CASE DP_Step3 OF 
100://负极叠片，正极在取片位
	bStandbyStep1_1:=FALSE;
	bStandbyStep1_2:=FALSE;
	DP_Step3:=110; 
110:   //叠负极片同时 判断证据能否取片  提高效率
	IF arrAxisCtrl[AxiseNo.VirAxisName.VirMain].Status.fActPos>=10  AND  arrAxisCtrl[AxiseNo.VirAxisName.VirMain].Status.fActPos<=220     THEN
	//正送片搬运极取片处理
		IF   arrAxisCtrl[AxiseNo.AxisName.AnCarryingUpDown].Cmd.arrbRealPoint[4] AND 
			  NOT Mach_Control.An_b.An_CarryingFalg    AND  ( Mach_Control.An_b.An_MainBeltOK OR  Mach_Control.U.EmptyRunMode )  AND 
			  NOT  Mach_Control.An_b.An_MainBelting   AND NOT  bStandbyStep1_1 AND (NOT An_JumpRules[3]  AND NOT  An_JumpRules[6] AND NOT An_JumpRules[8] AND NOT An_JumpRules[10])(*AND NOT Mach_Control.An_b.JumpPiceReady *) THEN
			   An_Step0:=10;//正极取流水线子程序
			   bStandbyStep1_1:=TRUE;
		END_IF
		
		IF arrAxisCtrl[AxiseNo.AxisName.AnDTCarryingUpDown].Cmd.arrbRealPoint[4] AND 
		 Mach_Control.An_b.An_deviationDPOK AND NOT Mach_Control.An_b.An_DPCarryingFalg AND  
			Mach_Control.An_b.An_deviationFalg  AND  NOT  bStandbyStep1_2  AND NOT DP_CheseCam  THEN
			An_Step3:=10;//正极取纠偏平台子程序
			bStandbyStep1_2:=TRUE;
		END_IF
	
	ELSIF  arrAxisCtrl[AxiseNo.VirAxisName.VirMain].Status.fActPos>220  THEN
		DP_Step3:=120;
	END_IF		   
	
	
120:
	arrCyCtrl[arrCyNo.ElectValveName.CadeviationVacuum].Cmd.bON:=TRUE;//负极纠偏平台真空开			
	arrCyCtrl[arrCyNo.ElectValveName.CadeviationVacuum].Cmd.bOFF:=FALSE;//负极纠偏平台真空开					
	IF 	arrAxisCtrl[AxiseNo.VirAxisName.VirMain].Status.fActPos>=234 THEN//198
		
		Mach_Control.Ca_b.Ca_Rectifydev_CS:=0;
		CCD.Over.Start.stPoleNo:=Par.stDT_date.Ca_MQ_Slice[8].stPoleNo;
		arrCyCtrl[arrCyNo.ElectValveName.CaDTCarryingVacuum].Cmd.bON:=TRUE;//负极叠片搬运真空破
		arrCyCtrl[arrCyNo.ElectValveName.CaDTCarryingVacuum].Cmd.bOFF:=FALSE;//负极叠片搬运真空破
		arrCyCtrl[arrCyNo.ElectValveName.CaCarryingVacuum2].Cmd.bON:=TRUE;//负极送片搬运真空破
		arrCyCtrl[arrCyNo.ElectValveName.CaCarryingVacuum2].Cmd.bOFF:=FALSE;//负极送片搬运真空破
		arrCyCtrl[arrCyNo.ElectValveName.CadeviationVacuum].Cmd.bON:=TRUE;//负极纠偏平台真空开
		arrCyCtrl[arrCyNo.ElectValveName.CadeviationVacuum].Cmd.bOFF:=FALSE;//负极纠偏平台真空开			
		
		Mach_Control.Ca_b.Ca_DPCarryingFalg :=FALSE;//复位负极叠片搬运吸盘上有料标记
		//IF Mach_Control.Ca_b.Ca_CarryingFalg THEN
			Mach_Control.Ca_b.Ca_deviationFalg:=TRUE;//置位纠偏平台上有料标记
			Mach_Control.Ca_b.Ca_CarryingFalg:=FALSE;//复位负极送片搬运吸盘上有料标记
		//END_IF
		Par.stDT_date.Ca_MQ_Slice[8]:=Par.stDT_date.Ca_MQ_Slice[7];
		
	END_IF	
	IF 	arrAxisCtrl[AxiseNo.VirAxisName.VirMain].Status.fActPos>=342 THEN//198
     	CCD.Over.Start.iPliesNo:=UINT_TO_INT(Mach_Control.Ca_b.Ca_Quantited + Mach_Control.An_b.An_Quantited+1);	
		IF NOT Ca_Number THEN
			CCD.Over.Start.iPhotoDo:=1;
		ELSE
			CCD.Over.Start.iPhotoDo:=2;
		END_IF
		Mach_Control.DT_b.CDD_OverStart:=TRUE;
		DP_Step3:=121;
	 END_IF		
		
121:
	IF 	arrAxisCtrl[AxiseNo.VirAxisName.VirMain].Status.fActPos>=360 THEN//198
		arrCyCtrl[arrCyNo.ElectValveName.CaCarryingVacuum2].Cmd.bON:=FALSE;//负极送片搬运真空开
		arrCyCtrl[arrCyNo.ElectValveName.CaCarryingVacuum2].Cmd.bOFF:=TRUE;//负极送片搬运真空开
		arrCyCtrl[arrCyNo.ElectValveName.CaDTCarryingVacuum].Cmd.bON:=FALSE;//负极叠片搬运真空破
		arrCyCtrl[arrCyNo.ElectValveName.CaDTCarryingVacuum].Cmd.bOFF:=TRUE;//负极叠片搬运真空破
		DP_Step3:=6666;
	END_IF	
	
	
200://负极叠片，正极在取片位

	IF iAnCamInSel2=1 THEN
		arrCyCtrl[arrCyNo.ElectValveName.AnDTCarryingVacuum].Cmd.bON:=TRUE;//正极送片搬运真空关
		arrCyCtrl[arrCyNo.ElectValveName.AnDTCarryingVacuum].Cmd.bOFF:=FALSE;//正极送片搬运真空关
	END_IF
	
	//fbAnDTCarryingVacuum.Vacuumsel:=SEL(iAnCamInSel2=1,0,1)     ;//	正极叠片搬运真空开	
	IF arrAxisCtrl[AxiseNo.VirAxisName.VirMain].Status.fActPos>=210 THEN//复检提前
		IF Mach_Control.DT_b.DT_CCD_TwoModel THEN												
			CCD.AnRec.Finish.RectifyResult:=0;
			CCD.AnRec.Finish.RectifyX1:=0;
			CCD.AnRec.Finish.RectifyX2:=0;
			CCD.AnRec.Finish.RectifyY:=0;												
			Mach_Control.An_b.An_CCDStart :=TRUE;//启动CCD拍照
			CCD.AnRec.Start.iPhotoDo:=2;//第二次拍照	
		END_IF
		DP_Step3:=205;
	END_IF
205:			
	IF NOT DP_CheseCam  AND NOT  An_JumpRules[3]  AND NOT  An_JumpRules[6] AND NOT An_JumpRules[8] AND NOT An_JumpRules[10] THEN
	
		IF arrAxisCtrl[AxiseNo.VirAxisName.VirMain].Status.fActPos>=225  AND arrAxisCtrl[AxiseNo.VirAxisName.VirMain].Status.fActPos<=230 THEN	
			//fbAnCamInCarryingUpDown.bCamInExecute:=FALSE;//正极升解除耦合															
			//fbAnCamInCarryingWhirling.bCamInExecute:=FALSE;//正极旋转解除耦合			
			//Mach_Control.An_b.An_MainBelting:=FALSE;//正极搬运升降取极片中																					
			IF  NOT  Mach_Control.Ca_b.Ca_deviationFPOK  THEN    //负极放片纠偏太未在初始位置报警  
					Mach_Control.Ca_b.Error_tips[1]:=TRUE ;
			END_IF											
			IF  NOT  Mach_Control.An_b.An_deviationDPOK  THEN    //正极取片纠偏未完成报警
					Mach_Control.An_b.Error_tips[1]:=TRUE;
			END_IF			
			IF Mach_Control.An_b.An_deviationDPOK OR Mach_Control.U.EmptyRunMode OR	TRUE  THEN // 
				arrCyCtrl[arrCyNo.ElectValveName.AnDTCarryingVacuum].Cmd.bON:=TRUE;//正极叠片搬运真空开	
				arrCyCtrl[arrCyNo.ElectValveName.AnDTCarryingVacuum].Cmd.bOFF:=FALSE;//正极叠片搬运真空开		
				An_deviationDPOKFalg:=TRUE;	
			ELSE		
				arrCyCtrl[arrCyNo.ElectValveName.AnDTCarryingVacuum].Cmd.bON:=FALSE;//正极叠片搬运真空开					
				arrCyCtrl[arrCyNo.ElectValveName.AnDTCarryingVacuum].Cmd.bOFF:=TRUE;//正极叠片搬运真空开												
				fbAnCamInDTCarryingUpDown.bCamInExecute:=FALSE;	//正极叠片搬运升降凸轮解耦				
				IF NOT arrAxisCtrl[AxiseNo.AxisName.AnDTCarryingUpDown].Cmd.arrbRealPoint[4]    THEN
						arrAxisCtrl[AxiseNo.AxisName.AnDTCarryingUpDown].Cmd.iGoSetPos:=4;   //到等待位
				END_IF			
			END_IF	
			//IF NOT Mach_Control.An_b.JumpPiceReady THEN
				An_Step0:=10;//调用正极取片程序	
			//END_IF
			DP_Step3:=210;														
		END_IF									
	ELSE
			DP_Step3:=210;	
	END_IF


210:
	//打开或关闭真空，标记对应位置有料
	IF 	arrAxisCtrl[AxiseNo.VirAxisName.VirMain].Status.fActPos>=234 THEN//198
	
		Mach_Control.Ca_b.Ca_Rectifydev_CS:=0;
		arrCyCtrl[arrCyNo.ElectValveName.CaCarryingVacuum2].Cmd.bON:=TRUE;//负极送片搬运真空关
		arrCyCtrl[arrCyNo.ElectValveName.CaCarryingVacuum2].Cmd.bOFF:=FALSE;//负极送片搬运真空关
		arrCyCtrl[arrCyNo.ElectValveName.CaDTCarryingVacuum].Cmd.bON:=TRUE;//负极叠片搬运直空关
		arrCyCtrl[arrCyNo.ElectValveName.CaDTCarryingVacuum].Cmd.bOFF:=FALSE;//负极叠片搬运直空关
		arrCyCtrl[arrCyNo.ElectValveName.CadeviationVacuum].Cmd.bON:=TRUE;//负极纠偏平台真空开	
		arrCyCtrl[arrCyNo.ElectValveName.CadeviationVacuum].Cmd.bOFF:=FALSE;//负极纠偏平台真空开		
		
		Mach_Control.Ca_b.Ca_DPCarryingFalg :=FALSE;//复位负极叠片搬运吸盘上有料标记
		//IF Mach_Control.Ca_b.Ca_CarryingFalg THEN
			Mach_Control.Ca_b.Ca_deviationFalg:=TRUE;//置位纠偏平台上有料标记
			Mach_Control.Ca_b.Ca_CarryingFalg:=FALSE;//复位负极送片搬运吸盘上有料标记
		//END_IF
		Par.stDT_date.Ca_MQ_Slice[8]:=Par.stDT_date.Ca_MQ_Slice[7];
		IF An_deviationDPOKFalg AND  iAnCamInSel2=1   THEN
			Par.stDT_date.An_MQ_Slice[2]:=Par.stDT_date.An_MQ_Slice[1];
			//IF Mach_Control.An_b.An_deviationFalg THEN
				Mach_Control.An_b.An_DPCarryingFalg :=TRUE;//复位正极叠片搬运吸盘上有料标记										
				Mach_Control.An_b.An_deviationFalg:=FALSE;//置位纠偏平台上有料标记	
			//END_IF										
			arrCyCtrl[arrCyNo.ElectValveName.AndeviationVacuum].Cmd.bOFF:=TRUE;//正极纠偏平台真空关
			arrCyCtrl[arrCyNo.ElectValveName.AndeviationVacuum].Cmd.bON:=FALSE;//正极纠偏平台真空关
			arrCyCtrl[arrCyNo.ElectValveName.AndeviationVacuumBark].Cmd.bON:=TRUE;//正极纠偏平台破真空开	
			arrCyCtrl[arrCyNo.ElectValveName.AndeviationVacuumBark].Cmd.bOFF:=FALSE;//正极纠偏平台破真空开	
	(*	
		ELSIF NOT   DP_CheseCam THEN								
			An_Step3:=10;//正极叠片搬运取纠偏台极片	
	*)																					
		END_IF
	
	END_IF

	IF 	arrAxisCtrl[AxiseNo.VirAxisName.VirMain].Status.fActPos>=342 THEN//198
		CCD.Over.Start.iPliesNo:=UINT_TO_INT(Mach_Control.Ca_b.Ca_Quantited + Mach_Control.An_b.An_Quantited+1);
		CCD.Over.Start.stPoleNo:=Par.stDT_date.Ca_MQ_Slice[8].stPoleNo;
		IF NOT Ca_Number THEN
			CCD.Over.Start.iPhotoDo:=1;
		ELSE
			CCD.Over.Start.iPhotoDo:=2;
		END_IF
		Mach_Control.DT_b.CDD_OverStart:=TRUE;	
		IF NOT Ca_Number THEN
			DP_Step3:=211;					
		END_IF	
    END_IF	
211:
	IF 	arrAxisCtrl[AxiseNo.VirAxisName.VirMain].Status.fActPos>=360 THEN//198	
		arrCyCtrl[arrCyNo.ElectValveName.CaCarryingVacuum2].Cmd.bON:=FALSE;//负极送片搬运真空开
		arrCyCtrl[arrCyNo.ElectValveName.CaCarryingVacuum2].Cmd.bOFF:=TRUE;//负极送片搬运真空开
		arrCyCtrl[arrCyNo.ElectValveName.CaDTCarryingVacuum].Cmd.bON:=FALSE;//负极叠片搬运直空开
		arrCyCtrl[arrCyNo.ElectValveName.CaDTCarryingVacuum].Cmd.bOFF:=TRUE;//负极叠片搬运直空开
		DP_Step3:=6666;					
	END_IF
			



		
300://正极叠片，负极在取片位			
	bStandbyStep1_3:=FALSE;
	bStandbyStep1_4:=FALSE;
	DP_Step3:=310; 		
310:	
	IF arrAxisCtrl[AxiseNo.VirAxisName.VirMain].Status.fActPos>=10  AND  arrAxisCtrl[AxiseNo.VirAxisName.VirMain].Status.fActPos<=220     THEN
		//正送片搬运极取片处理
		IF   arrAxisCtrl[AxiseNo.AxisName.CaCarryingUpDown2].Cmd.arrbRealPoint[4] AND 
			NOT Mach_Control.Ca_b.Ca_CarryingFalg    AND  ( Mach_Control.Ca_b.Ca_CacheBeltDLOK OR  Mach_Control.U.EmptyRunMode )  AND 
			NOT  Mach_Control.Ca_b.Ca_CacheBelting   AND NOT  bStandbyStep1_3 THEN
			Ca_Step0:=10;   //负极取流水线子程序
			bStandbyStep1_3:=TRUE;
		END_IF
	
		IF arrAxisCtrl[AxiseNo.AxisName.CaDTCarryingUpDown].Cmd.arrbRealPoint[4] AND 
			Mach_Control.Ca_b.Ca_deviationDPOK AND NOT Mach_Control.Ca_b.Ca_DPCarryingFalg AND  
			Mach_Control.Ca_b.Ca_deviationFalg AND  NOT  bStandbyStep1_4   THEN
			Ca_Step3:=10;     //负极取纠偏平台子程序
			bStandbyStep1_4:=TRUE;
		END_IF					
	ELSIF  arrAxisCtrl[AxiseNo.VirAxisName.VirMain].Status.fActPos>220  THEN
			DP_Step3:=320; 
	END_IF	
	
320://正极叠片，负极在取片位
	arrCyCtrl[arrCyNo.ElectValveName.AndeviationVacuum].Cmd.bON:=TRUE;//正极纠偏平台真空开			
	arrCyCtrl[arrCyNo.ElectValveName.AndeviationVacuum].Cmd.bOFF:=FALSE;//正极纠偏平台真空开					
	IF 	arrAxisCtrl[AxiseNo.VirAxisName.VirMain].Status.fActPos>=234 THEN//198
	
		Mach_Control.An_b.An_Rectifydev_CS:=0;	
		arrCyCtrl[arrCyNo.ElectValveName.AnCarryingVacuum].Cmd.bON:=FALSE;//正极送片搬运真空关
		arrCyCtrl[arrCyNo.ElectValveName.AnCarryingVacuum].Cmd.bOFF:=TRUE;//正极送片搬运真空关
		arrCyCtrl[arrCyNo.ElectValveName.AnCarryingVacuumBark].Cmd.bON:=TRUE;//正极送片搬运破真空开
		arrCyCtrl[arrCyNo.ElectValveName.AnCarryingVacuumBark].Cmd.bOFF:=FALSE;//正极送片搬运破真空开
		
		arrCyCtrl[arrCyNo.ElectValveName.AnDTCarryingVacuum].Cmd.bON:=FALSE;//正极送片搬运真空关
		arrCyCtrl[arrCyNo.ElectValveName.AnDTCarryingVacuum].Cmd.bOFF:=TRUE;//正极送片搬运真空关
		arrCyCtrl[arrCyNo.ElectValveName.AnDTCarryingVacuumBark].Cmd.bON:=TRUE;//正极送片搬运破真空开
		arrCyCtrl[arrCyNo.ElectValveName.AnDTCarryingVacuumBark].Cmd.bOFF:=FALSE;//正极送片搬运破真空开
		
		arrCyCtrl[arrCyNo.ElectValveName.AndeviationVacuum].Cmd.bON:=TRUE;//正极纠偏平台真空开		
		arrCyCtrl[arrCyNo.ElectValveName.AndeviationVacuum].Cmd.bOFF:=FALSE;//正极纠偏平台真空开		
		
		
		Mach_Control.An_b.An_DPCarryingFalg :=FALSE;//复位正极叠片搬运吸盘上有料标记
		//IF Mach_Control.An_b.An_CarryingFalg THEN
			Mach_Control.An_b.An_deviationFalg:=TRUE;//置位纠偏平台上有料标记
			Mach_Control.An_b.An_CarryingFalg:=FALSE;//复位正极送片搬运吸盘上有料标记
		//END_IF
		Par.stDT_date.An_MQ_Slice[1]:=Par.stDT_date.An_MQ_Slice[0];
		
	END_IF
	
	IF 	arrAxisCtrl[AxiseNo.VirAxisName.VirMain].Status.fActPos>=342 THEN//198
		CCD.Over.Start.iPliesNo:=UINT_TO_INT(Mach_Control.Ca_b.Ca_Quantited + Mach_Control.An_b.An_Quantited+1);
		CCD.Over.Start.stPoleNo:=Par.stDT_date.An_MQ_Slice[2].stPoleNo;
		IF NOT An_Number THEN
			CCD.Over.Start.iPhotoDo:=1;
		ELSE
			CCD.Over.Start.iPhotoDo:=2;
		END_IF
		Mach_Control.DT_b.CDD_OverStart:=TRUE;				
		DP_Step3:=6666;	
	END_IF
400:	//复检提前------//正极叠片，负极在叠片位

	//fbCaDTCarryingVacuum.Vacuumsel:= SEL(iCaCamInSel2=1 ,0,1)   ;//	负极叠片搬运真空开
	IF iCaCamInSel2=1 THEN
		arrCyCtrl[arrCyNo.ElectValveName.CaDTCarryingVacuum].Cmd.bON:=FALSE;//负极叠台搬运真空开	
		arrCyCtrl[arrCyNo.ElectValveName.CaDTCarryingVacuum].Cmd.bOFF:=TRUE;//负极叠台搬运真空开		
	END_IF

	IF 	arrAxisCtrl[AxiseNo.VirAxisName.VirMain].Status.fActPos>=210 THEN//198
		IF Mach_Control.DT_b.DT_CCD_TwoModel THEN
				CCD.CaRec.Finish.RectifyX1:=0;
				CCD.CaRec.Finish.RectifyX2:=0;
				CCD.CaRec.Finish.RectifyY:=0;		
				CCD.CaRec.Finish.RectifyResult:=0;//拍照结果清零									
				Mach_Control.Ca_b.Ca_CCDStart :=TRUE;//启动CCD拍照
				CCD.CaRec.Start.iPhotoDo:=2;//启动CCD第二次拍照									
		END_IF
		DP_Step3:=405;
	END_IF
405:		
	IF arrAxisCtrl[AxiseNo.VirAxisName.VirMain].Status.fActPos>=225  AND arrAxisCtrl[AxiseNo.VirAxisName.VirMain].Status.fActPos<=230 THEN																								
		IF  NOT  Mach_Control.An_b.An_deviationFPOK  THEN    //正极放片纠偏太未在初始位置报警  
			  Mach_Control.An_b.Error_tips[2]:=TRUE ;
		END_IF
		
		IF  NOT  Mach_Control.Ca_b.Ca_deviationDPOK  THEN    //负极取片纠偏未完成报警
			  Mach_Control.Ca_b.Error_tips[2]:=TRUE ;
		END_IF		

		//正极叠片时平移到位后判断正极纠偏台是否允许放片
		IF Mach_Control.An_b.An_deviationFPOK OR Mach_Control.U.EmptyRunMode  THEN 
				An_deviationFPOKFalg:=TRUE;//正极纠偏平台允许放片标记
		ELSE									
			fbAnCamInCarryingUpDown.bCamInExecute:=FALSE;	//正极送片搬运升降凸轮解耦				
			IF NOT arrAxisCtrl[AxiseNo.AxisName.AnCarryingUpDown].Cmd.arrbRealPoint[4]    THEN
				arrAxisCtrl[AxiseNo.AxisName.AnCarryingUpDown].Cmd.iGoSetPos:=4;
			END_IF;				
		END_IF					
		IF Mach_Control.Ca_b.Ca_deviationDPOK OR Mach_Control.U.EmptyRunMode OR TRUE  THEN //  
			Ca_deviationDPOKFalg:=TRUE;	
			arrCyCtrl[arrCyNo.ElectValveName.CaDTCarryingVacuum].Cmd.bON:=FALSE;//负极叠片搬运真空开	
			arrCyCtrl[arrCyNo.ElectValveName.CaDTCarryingVacuum].Cmd.bOFF:=TRUE;//负极叠片搬运真空开		
		ELSE	
			//arrCyCtrl[arrCyNo.ElectValveName.CaDTCarryingVacuum].Cmd.bON:=FALSE;//负极叠片搬运真空开									
			fbCaCamInDTCarryingUpDown.bCamInExecute:=FALSE;	//负极叠片搬运升降凸轮解耦				
			IF NOT arrAxisCtrl[AxiseNo.AxisName.CaDTCarryingUpDown].Cmd.arrbRealPoint[4]    THEN
				arrAxisCtrl[AxiseNo.AxisName.CaDTCarryingUpDown].Cmd.iGoSetPos:=4;   //到等待位
			ELSE
				arrAxisCtrl[AxiseNo.AxisName.CaDTCarryingUpDown].Cmd.iGoSetPos:=0;   //到等待位
			END_IF;				
		END_IF									
		Ca_Step0:=10;//调用负极取片程序       取片允许条件在子程序里
		DP_Step3:=410;		
	END_IF
(*	
	//判断是否允许负极送片搬运取料
	IF arrAxisCtrl[AxiseNo.VirAxisName.VirMain].Status.fActPos>=CamOutArgel  AND arrAxisCtrl[AxiseNo.VirAxisName.VirMain].Status.fActPos<=(CamOutArgel+5) THEN
		IF (Mach_Control.Ca_b.Ca_CacheBeltDLOK AND NOT fbCaCamInCarryingUpDown2OutCamFlge) OR Mach_Control.U.EmptyRunMode  THEN
			Mach_Control.Ca_b.Ca_CacheBelting:=TRUE;//f负极搬运升降取极片中	
			arrCyCtrl[arrCyNo.ElectValveName.CaCarryingVacuum2].Cmd.bON:=FALSE;//负极送片搬运真空开
			arrCyCtrl[arrCyNo.ElectValveName.CaCarryingVacuum2].Cmd.bOFF:=TRUE;//负极送片搬运真空开
		ELSE
			//arrCyCtrl[arrCyNo.ElectValveName.CaCarryingVacuum2].Cmd.bON:=FALSE;//负极送片搬运真空开
			fbCaCamInCarryingUpDown2.bCamInExecute:=FALSE;//负极升解除耦合
			Mach_Control.Ca_b.Ca_CacheBelting:=FALSE;
		END_IF								
	END_IF
	//解除负极搬运升降凸轮耦合标记
	fbCaCamInCarryingUpDown2OutCam_F_TRIG(CLK:=fbCaCamInCarryingUpDown2.bCamInExecute , Q=> );
	IF fbCaCamInCarryingUpDown2OutCam_F_TRIG.Q THEN
		fbCaCamInCarryingUpDown2OutCamFlge:=TRUE;//负极升降2凸轮解耦标记
	END_IF	
*)			
410:							
	//打开或关闭真空，标记对应位置有料
	IF 	arrAxisCtrl[AxiseNo.VirAxisName.VirMain].Status.fActPos>=234 THEN//198

		Mach_Control.An_b.An_Rectifydev_CS:=0;
		CCD.Over.Start.stPoleNo:=Par.stDT_date.An_MQ_Slice[2].stPoleNo;
	(*	
		arrCyCtrl[arrCyNo.ElectValveName.AnCarryingVacuum].Cmd.bOFF:=TRUE;//正极送片搬运真空关
		arrCyCtrl[arrCyNo.ElectValveName.AnCarryingVacuumBark].Cmd.bON:=TRUE;//正极送片搬运破真空开
		arrCyCtrl[arrCyNo.ElectValveName.AnDTCarryingVacuum].Cmd.bOFF:=TRUE;//正极叠片搬运真空关
		arrCyCtrl[arrCyNo.ElectValveName.AnDTCarryingVacuumBark].Cmd.bON:=TRUE;//正极叠片搬运破真空开
	*)	
		arrCyCtrl[arrCyNo.ElectValveName.AnCarryingVacuum].Cmd.bON:=FALSE;//正极送片搬运真空关
		arrCyCtrl[arrCyNo.ElectValveName.AnCarryingVacuum].Cmd.bOFF:=TRUE;//正极送片搬运真空关
		arrCyCtrl[arrCyNo.ElectValveName.AnCarryingVacuumBark].Cmd.bON:=TRUE;//正极送片搬运破真空开
		arrCyCtrl[arrCyNo.ElectValveName.AnCarryingVacuumBark].Cmd.bOFF:=FALSE;//正极送片搬运破真空开
		
		arrCyCtrl[arrCyNo.ElectValveName.AnDTCarryingVacuum].Cmd.bON:=FALSE;//正极送片搬运真空关
		arrCyCtrl[arrCyNo.ElectValveName.AnDTCarryingVacuum].Cmd.bOFF:=TRUE;//正极送片搬运真空关
		arrCyCtrl[arrCyNo.ElectValveName.AnDTCarryingVacuumBark].Cmd.bON:=TRUE;//正极送片搬运破真空开
		arrCyCtrl[arrCyNo.ElectValveName.AnDTCarryingVacuumBark].Cmd.bOFF:=FALSE;//正极送片搬运破真空开	
		
		arrCyCtrl[arrCyNo.ElectValveName.AndeviationVacuum].Cmd.bON:=TRUE;//正极纠偏平台真空开	
		arrCyCtrl[arrCyNo.ElectValveName.AndeviationVacuum].Cmd.bOFF:=FALSE;//正极纠偏平台真空开	

		Mach_Control.An_b.An_DPCarryingFalg :=FALSE;//复位正极叠片搬运吸盘上有料标记
		//IF Mach_Control.An_b.An_CarryingFalg THEN
			Mach_Control.An_b.An_deviationFalg:=TRUE;//置位纠偏平台上有料标记
			Mach_Control.An_b.An_CarryingFalg:=FALSE;//复位正极送片搬运吸盘上有料标记
		//END_IF
		
		Par.stDT_date.An_MQ_Slice[1]:=Par.stDT_date.An_MQ_Slice[0];
		
		(*
		IF (Mach_Control.Ca_b.Ca_CacheBelting AND NOT fbCaCamInCarryingUpDown2OutCamFlge) OR Mach_Control.U.EmptyRunMode  THEN
			Mach_Control.Ca_b.Ca_CarryingFalg:=TRUE;//复位负极送片搬运吸盘上有料标记
			Par.stDT_date.Ca_MQ_Slice[7]:=Par.stDT_date.Ca_MQ_Slice[6];
		END_IF*)
		
		
		arrAxisCtrl[AxiseNo.AxisName.CaCarryingUpDown2].Cmd.bStop:=FALSE;
	

		//判断负极纠偏台是否允许取料
		IF Ca_deviationDPOKFalg AND NOT DP_CheseCam AND iCaCamInSel2=1 THEN		
			arrCyCtrl[arrCyNo.ElectValveName.CaDTCarryingVacuum].Cmd.bON:=FALSE;//负极叠台搬运真空开	
			arrCyCtrl[arrCyNo.ElectValveName.CaDTCarryingVacuum].Cmd.bOFF:=TRUE;//负极叠台搬运真空开	
			arrCyCtrl[arrCyNo.ElectValveName.CadeviationVacuum].Cmd.bOFF:=TRUE;//负极纠偏平台真空关
			arrCyCtrl[arrCyNo.ElectValveName.CadeviationVacuum].Cmd.bON:=FALSE;//负极纠偏平台真空关
			arrCyCtrl[arrCyNo.ElectValveName.CadeviationVacuumBark].Cmd.bON:=TRUE;//负极纠偏平台破真空开	
			arrCyCtrl[arrCyNo.ElectValveName.CadeviationVacuumBark].Cmd.bOFF:=FALSE;//负极纠偏平台破真空开		
			//IF 	Mach_Control.Ca_b.Ca_deviationFalg THEN				
				Mach_Control.Ca_b.Ca_DPCarryingFalg :=TRUE;//置位负极叠片搬运吸盘上有料标记			
				Mach_Control.Ca_b.Ca_deviationFalg:=FALSE;//复位负极纠偏平台上有料标记	
			//END_IF			
			Par.stDT_date.Ca_MQ_Slice[9]:=Par.stDT_date.Ca_MQ_Slice[8];
		(*	
		ELSE   
			Ca_Step3:=10;//负极叠片搬运取纠偏台极片	
		*)	   
		END_IF									

		//判断正极纠偏台是否允许放料
		IF An_deviationFPOKFalg THEN			
			arrCyCtrl[arrCyNo.ElectValveName.AnCarryingVacuumBark].Cmd.bON:=TRUE;//正极送片搬运真空关
			arrCyCtrl[arrCyNo.ElectValveName.AnCarryingVacuumBark].Cmd.bOFF:=FALSE;//正极送片搬运破真空开
			arrCyCtrl[arrCyNo.ElectValveName.AndeviationVacuum].Cmd.bON:=TRUE;//正极纠偏平台真空开		
			arrCyCtrl[arrCyNo.ElectValveName.AndeviationVacuum].Cmd.bOFF:=FALSE;//正极纠偏平台真空开	
			//IF Mach_Control.An_b.An_CarryingFalg THEN	
				Mach_Control.An_b.An_deviationFalg:=TRUE;//置位正极纠偏平台上有料标记
				Mach_Control.An_b.An_CarryingFalg:=FALSE;//复位正极送片搬运吸盘上有料标记						
			//END_IF			
			Par.stDT_date.An_MQ_Slice[1]:=Par.stDT_date.An_MQ_Slice[0];//送片机械手传送至纠偏平台
		ELSE   
			An_Step1:=10;//正极送片搬运放片到纠偏台			   
		END_IF
	END_IF

		IF 	arrAxisCtrl[AxiseNo.VirAxisName.VirMain].Status.fActPos>=342 THEN//198
			CCD.Over.Start.iPliesNo:=UINT_TO_INT(Mach_Control.Ca_b.Ca_Quantited + Mach_Control.An_b.An_Quantited+1);	
			IF NOT An_Number THEN
				CCD.Over.Start.iPhotoDo:=1;
			ELSE
				CCD.Over.Start.iPhotoDo:=2;
			END_IF
			CCD.Over.Finish.OverhandResult:=0;
			Mach_Control.DT_b.CDD_OverStart:=TRUE;	
			IF NOT An_Number THEN
				DP_Step3:=6666;					
			END_IF
			
        END_IF
END_CASE



//判断主轴是否完成
CASE  DP_Step4 OF
100://叠负极主轴定位完成判断				
	IF arrAxis[AxiseNo.VirAxisName.VirMain].NcToPlc.SetPos=360 AND  arrAxis[AxiseNo.VirAxisName.VirMain].Status.NotMoving  THEN
		//如果，叠片搬运掉片报警就不计数		
		IF NOT Ca_Number THEN
			Mach_Control.Ca_b.Ca_Quantited:=Mach_Control.Ca_b.Ca_Quantited+1;
			DPcount:=DPcount+1;
			IF Mach_Control.U.EmptyRunMode THEN
				Mach_Control.Ca_b.Ca_EmptyRunKDQuantited:=Mach_Control.Ca_b.Ca_EmptyRunKDQuantited +1;
//			ELSE
//				Mach_Control.Ca_b.Ca_EmptyRunKDQuantited:=0;
			END_IF
			Par.stDT_date.YD_JS_L:=Par.stDT_date.YD_JS_L+1;
			Mach_Control.Ca_b.Ca_CCD_amount:=0;
				//叠台升降轴下降
				IF NOT Mach_Control.U.EmptyRunMode  THEN
					arrAxisCtrl[AxiseNo.AxisName.DTUpDown].Cmd.fPosition_of_Rel:=-(Par.stDT_date.Ca_Thickness+Par.stDT_date.SEPTA_Thickness+Par.stDT_date.Pole_ThicknessCom);
				ELSE
					arrAxisCtrl[AxiseNo.AxisName.DTUpDown].Cmd.fPosition_of_Rel:=-Par.stDT_date.SEPTA_Thickness;
				END_IF
				IF Mach_Control.Ca_b.Ca_Quantited + Mach_Control.An_b.An_Quantited>3 THEN
					arrAxisPar[AxiseNo.AxisName.DTUpDown].fVelocity_of_Rel:=100;
					arrAxisCtrl[AxiseNo.AxisName.DTUpDown].Cmd.bMoveRel:=TRUE;
				END_IF
		END_IF
		Mach_Control.An_b.An_CCDStart :=FALSE;//启动CCD拍照						
		DP_Step1:=100;//解除耦合，主轴回零子程序
		
		IF Mach_Control.DT_b.SinStepMode THEN//单步调试模式
			DP_SinStepe:=TRUE;
		ELSE
			DP_SinStepe:=FALSE;	
		END_IF
		
		DP_Step0:=0;
		Ca_AlarmTON[11].IN:=FALSE;
		IF Ca_Number  THEN
			DP_Step6:=6666;
		ELSIF Mach_Control.DT_b.DT_Overhang THEN
			DP_Step6:=102;
		ELSE
			DP_Step6:=101;
		END_IF	
		DP_Step4:=110;	
	END_IF;	
110:
	IF ((*Ca_deviationFPOKFalg OR*) Ca_Step1=6666 OR Ca_Step1=0) AND ((*An_deviationDPOKFalg OR *)An_Step3=6666 OR An_Step3=0)  
		AND ((An_Step0=6666 OR An_Step0=0) OR Mach_Control.An_b.An_Quantited=Par.stDT_date.An_Quantity )  THEN         
		DP_Step4:=6666;
		DP_Step0:=0;
		Ca_deviationFPOKFalg:=FALSE;
		An_deviationDPOKFalg:=FALSE;  
	END_IF



		
200:	//叠正极主轴定位完成判断
	IF arrAxis[AxiseNo.VirAxisName.VirMain].NcToPlc.SetPos>=200 AND  NOT fbCaCamInCarryingUpDown2.bCamInExecute  THEN
		(*
		IF NOT  arrAxisCtrl[AxiseNo.AxisName.CaCarryingUpDown2].Cmd.arrbRealPoint[4] THEN
			arrAxisCtrl[AxiseNo.AxisName.CaCarryingUpDown2].Cmd.iGoSetPos:=4;//移动至流水线上方
		ELSE
			arrAxisCtrl[AxiseNo.AxisName.CaCarryingUpDown2].Cmd.iGoSetPos:=0;//移动至流水线上方
		END_IF
		*)
		;
	END_IF
	
	IF arrAxis[AxiseNo.VirAxisName.VirMain].NcToPlc.SetPos=360 AND  arrAxis[AxiseNo.VirAxisName.VirMain].Status.NotMoving  THEN
		//如果，叠片搬运掉片报警就不计数				
		IF NOT An_Number THEN
			Mach_Control.An_b.An_Quantited:=Mach_Control.An_b.An_Quantited+1;
			DPcount:=DPcount+1;			
			IF Mach_Control.U.EmptyRunMode THEN
				Mach_Control.An_b.An_EmptyRunKDQuantited:=Mach_Control.An_b.An_EmptyRunKDQuantited +1;
//			ELSE
//				Mach_Control.An_b.An_EmptyRunKDQuantited:=0;
			END_IF
			Par.stDT_date.YD_JS_R:=Par.stDT_date.YD_JS_R+1;
			Mach_Control.An_b.An_CCD_amount:=0;
			//叠台升降轴下降
			IF NOT Mach_Control.U.EmptyRunMode  THEN
					arrAxisCtrl[AxiseNo.AxisName.DTUpDown].Cmd.fPosition_of_Rel:=-(Par.stDT_date.An_Thickness+Par.stDT_date.SEPTA_Thickness+Par.stDT_date.Pole_ThicknessCom);
			ELSE
					arrAxisCtrl[AxiseNo.AxisName.DTUpDown].Cmd.fPosition_of_Rel:=-Par.stDT_date.SEPTA_Thickness;
			END_IF
			IF Mach_Control.Ca_b.Ca_Quantited + Mach_Control.An_b.An_Quantited>3 THEN
					arrAxisPar[AxiseNo.AxisName.DTUpDown].fVelocity_of_Rel:=100;
					arrAxisCtrl[AxiseNo.AxisName.DTUpDown].Cmd.bMoveRel:=TRUE;
			END_IF	
		END_IF
		Mach_Control.Ca_b.Ca_CCDStart :=FALSE;//启动CCD拍照			
		DP_Step1:=100;//解除耦合，主轴回零	

		(*
		IF  (Mach_Control.Ca_b.Ca_CacheBelting AND NOT fbCaCamInCarryingUpDown2OutCamFlge) OR Mach_Control.U.EmptyRunMode  THEN
			Par.stDT_date.Ca_betlCount.5:=FALSE;//复位负极流水线极片标记
			Mach_Control.Ca_b.Ca_CacheBelting:=FALSE;
		END_IF	*)
	
						
		arrCyCtrl[arrCyNo.ElectValveName.CadeviationVacuumBark].Cmd.bOFF:=TRUE;//负极纠偏平台破真空关	
		IF Mach_Control.DT_b.SinStepMode THEN//单步调试模式
			DP_SinStepe:=TRUE;
		ELSE
			DP_SinStepe:=FALSE;	
		END_IF							
		DP_Step0:=0;
		An_AlarmTON[11].IN:=FALSE;
		IF An_Number THEN
			  DP_Step7:=6666;
		ELSIF  Mach_Control.DT_b.DT_Overhang THEN
			  DP_Step7:=202;
		ELSE
			  DP_Step7:=201;
		END_IF
		DP_Step4:=210;	
		(*	
			IF  Mach_Control.DT_b.DT_Overhang AND NOT An_Number THEN
				  DP_Step7:=202;
			ELSIF An_Number THEN
				  DP_Step7:=6666;
			ELSE
				  DP_Step7:=201;
			END_IF
			DP_Step4:=6666;	
		*)
	END_IF;	
210:
	IF ((*An_deviationFPOKFalg OR *)An_Step1=6666 OR An_Step1=0) AND ((*Ca_deviationDPOKFalg OR *)Ca_Step3=6666 OR Ca_Step3=0) 
	AND (Ca_Step0=6666 OR Ca_Step0=0) THEN          
		DP_Step4:=6666;
		DP_Step0:=0;
		An_deviationFPOKFalg:=FALSE;
		Ca_deviationDPOKFalg:=FALSE; 
	END_IF

			
END_CASE



//观察NG片用，发现问题后删除
IF Ca_NGTest1.Q THEN
	Ca_NG:=Ca_NG+1;
END_IF


CASE  DP_Step5 OF
100://判断主轴运行时负极叠片搬运升降真空报警
	IF arrAxisCtrl[AxiseNo.VirAxisName.VirMain].Status.fActPos>0 AND arrAxisCtrl[AxiseNo.VirAxisName.VirMain].Status.fActPos<220 THEN
		IF Ca_Number THEN	
			DP_Step5:=110;
			arrCyCtrl[arrCyNo.ElectValveName.CaDTCarryingVacuum].Cmd.bON:=TRUE;//负极叠片搬运破真空开	
			arrCyCtrl[arrCyNo.ElectValveName.CaDTCarryingVacuum].Cmd.bOFF:=FALSE;//负极叠片搬运破真空开	
		END_IF
		Ca_NGTest1(CLK:=(CCD.CaRec.Finish.RectifyResult=2) , Q=> );
	ELSE 
		DP_Step5:=6666;
	END_IF

110:
	fbCaCamInDTCarryingUpDown.bCamInExecute:=FALSE;//负极叠片搬运升降
	fbCamInLeftYDUpDown.bCamInExecute:=FALSE;//左压刀升降
	fbCamInLeftYDLine.bCamInExecute:=FALSE;//左压刀开合
	IF NOT  fbCaCamInDTCarryingUpDown.bCamInExecute AND NOT fbCamInLeftYDUpDown.bCamInExecute AND NOT  fbCamInLeftYDLine.bCamInExecute THEN
		DP_Step5:=120;
		arrCyCtrl[arrCyNo.ElectValveName.CaDTCarryingVacuum].Cmd.bON:=FALSE;//负极叠片搬运真空开
		arrCyCtrl[arrCyNo.ElectValveName.CaDTCarryingVacuum].Cmd.bOFF:=TRUE;//负极叠片搬运真空开
	END_IF

120:
	arrAxisCtrl[AxiseNo.AxisName.CaDTCarryingUpDown].Cmd.bGearOut:=TRUE;
	arrAxisCtrl[AxiseNo.AxisName.LeftYDLine].Cmd.bGearOut:=TRUE;
	arrAxisCtrl[AxiseNo.AxisName.LeftYDUpDown].Cmd.bGearOut:=TRUE;
	IF NOT arrAxisCtrl[AxiseNo.AxisName.CaDTCarryingUpDown].Status.Coupled AND NOT arrAxisCtrl[AxiseNo.AxisName.LeftYDLine].Status.Coupled
	AND NOT arrAxisCtrl[AxiseNo.AxisName.LeftYDUpDown].Status.Coupled THEN
		arrAxisCtrl[AxiseNo.AxisName.CaDTCarryingUpDown].Cmd.bGearOut:=FALSE;
		arrAxisCtrl[AxiseNo.AxisName.LeftYDLine].Cmd.bGearOut:=FALSE;
		arrAxisCtrl[AxiseNo.AxisName.LeftYDUpDown].Cmd.bGearOut:=FALSE;
		DP_Step5:=130;
	END_IF

130:
	IF arrAxisCtrl[AxiseNo.AxisName.CaDTCarryingUpDown].Status.Homed AND arrAxisCtrl[AxiseNo.AxisName.CaDTCarryingUpDown].Status.NoMoving AND 
		NOT arrAxisCtrl[AxiseNo.AxisName.CaDTCarryingUpDown].Status.Error THEN
		IF arrAxisCtrl[AxiseNo.AxisName.CaDTCarryingUpDown].Cmd.arrbRealPoint[4] THEN
			arrCyCtrl[arrCyNo.ElectValveName.CaDTCarryingVacuum].Cmd.bON:=FALSE;//负极叠片搬运真空开
			arrCyCtrl[arrCyNo.ElectValveName.CaDTCarryingVacuum].Cmd.bOFF:=TRUE;//负极叠片搬运真空开
			arrAxisCtrl[AxiseNo.AxisName.CaDTCarryingUpDown].Cmd.iGoSetPos:=0;
			DP_Step5:=6666;
		ELSE
			arrAxisCtrl[AxiseNo.AxisName.CaDTCarryingUpDown].Cmd.iGoSetPos:=4;//负极叠片升降移动至等待高度
		END_IF
	END_IF







200://判断主轴运行时正极叠片搬运升降真空报警
	IF arrAxisCtrl[AxiseNo.VirAxisName.VirMain].Status.fActPos>0 AND arrAxisCtrl[AxiseNo.VirAxisName.VirMain].Status.fActPos<220 THEN
		IF An_Number THEN	
			DP_Step5:=210;
			arrCyCtrl[arrCyNo.ElectValveName.AnDTCarryingVacuumBark].Cmd.bON:=TRUE;//正极叠片搬运破真空开	
		END_IF
	ELSE 
		DP_Step5:=6666;
	END_IF

210:
	fbAnCamInDTCarryingUpDown.bCamInExecute:=FALSE;//正极叠片搬运升降
	fbCamInRightYDUpDown.bCamInExecute:=FALSE;
	fbCamInRightYDLine.bCamInExecute:=FALSE;
	IF NOT fbAnCamInDTCarryingUpDown.bCamInExecute AND NOT fbCamInRightYDUpDown.bCamInExecute AND NOT fbCamInRightYDLine.bCamInExecute THEN
		DP_Step5:=220;
		arrCyCtrl[arrCyNo.ElectValveName.AnDTCarryingVacuumBark].Cmd.bON:=FALSE;//正极叠片搬运破真空关	
	END_IF
220:
	arrAxisCtrl[AxiseNo.AxisName.AnDTCarryingUpDown].Cmd.bGearOut:=TRUE;
	arrAxisCtrl[AxiseNo.AxisName.RightYDLine].Cmd.bGearOut:=TRUE;
	arrAxisCtrl[AxiseNo.AxisName.RightYDUpDown].Cmd.bGearOut:=TRUE;
	IF NOT arrAxisCtrl[AxiseNo.AxisName.AnDTCarryingUpDown].Status.Coupled AND NOT arrAxisCtrl[AxiseNo.AxisName.RightYDLine].Status.Coupled AND
		NOT arrAxisCtrl[AxiseNo.AxisName.RightYDUpDown].Status.Coupled  THEN
		arrAxisCtrl[AxiseNo.AxisName.AnDTCarryingUpDown].Cmd.bGearOut:=FALSE;
		arrAxisCtrl[AxiseNo.AxisName.RightYDLine].Cmd.bGearOut:=FALSE;
		arrAxisCtrl[AxiseNo.AxisName.RightYDUpDown].Cmd.bGearOut:=FALSE;
		DP_Step5:=230;
	END_IF

230:
	IF arrAxisCtrl[AxiseNo.AxisName.AnDTCarryingUpDown].Status.Homed AND arrAxisCtrl[AxiseNo.AxisName.AnDTCarryingUpDown].Status.NoMoving AND 
	NOT arrAxisCtrl[AxiseNo.AxisName.AnDTCarryingUpDown].Status.Error THEN
		IF arrAxisCtrl[AxiseNo.AxisName.AnDTCarryingUpDown].Cmd.arrbRealPoint[4] THEN
			arrAxisCtrl[AxiseNo.AxisName.AnDTCarryingUpDown].Cmd.iGoSetPos:=0;
			DP_Step5:=6666;
		ELSE
			arrAxisCtrl[AxiseNo.AxisName.AnDTCarryingUpDown].Cmd.iGoSetPos:=4;//正极叠片升降移动至等待高度
		END_IF
	END_IF
		
END_CASE




CASE DP_Step6 OF
101:
	IF (CCD.Over.Finish.OverhandResult=4 OR CCD.Over.Finish.OverhandResult=2 OR CCD.Over.Finish.OverhandResult=1 ) AND NOT Ca_Number 
		AND( (arrAxisCtrl[AxiseNo.VirAxisName.VirMain].Status.fActPos>100 AND  arrAxisCtrl[AxiseNo.VirAxisName.VirMain].Status.fActPos<220) OR (arrAxisCtrl[AxiseNo.VirAxisName.VirMain].Status.fActPos=360)) THEN		
		DP_Step6:=102;
	ELSIF Ca_Number OR Mach_Control.U.EmptyRunMode OR Mach_Control.DT_b.DT_Overhang THEN//负极报警，空跑模式，Overhang屏蔽直接跳过
		DP_Step6:=6666;
	ELSIF NOT Ca_Number AND arrAxisCtrl[AxiseNo.VirAxisName.VirMain].Status.fActPos>220 AND arrAxisCtrl[AxiseNo.VirAxisName.VirMain].Status.fActPos<360 
		AND  CCD.Over.Finish.OverhandResult=0   THEN
		Mach_Control.Ca_b.Error[25]:=TRUE;//负极极片对齐度检测返回结果超时
		Par.stDT_date.Overhang_CSJS:=Par.stDT_date.Overhang_CSJS+1;
		DP_Step6:=6666;
	ELSIF CCD.Over.Finish.OverhandResult=3   THEN		
		Mach_Control.Ca_b.Error[27]:=TRUE;  //负极极片对齐度检测返回结果无片报警
		DP_Step6:=102;
	END_IF
					
102:
	CellMemory[Mach_Control.DT_b.DT_Memory].Overhang_Result[CCD.Over.Start.iPliesNo]:=CCD.Over.Finish.OverhandResult;
	CellMemory[Mach_Control.DT_b.DT_Memory].DiaphragmUnwindingTension2[CCD.Over.Start.iPliesNo]:=LIMIT(150,ABS(Mach_Control.DT_b.DiaphragmUnwindingTension),250);	
	CellMemory[Mach_Control.DT_b.DT_Memory].Ca_Ear_Overhang_A_C[Mach_Control.Ca_b.Ca_Quantited]:=ABS(CCD.Over.Finish.AnCaOverhandX1);
	CellMemory[Mach_Control.DT_b.DT_Memory].Ca_Ear_Overhang_S_CIL[Mach_Control.Ca_b.Ca_Quantited]:=ABS(CCD.Over.Finish.PoleOverhandX1);
	CellMemory[Mach_Control.DT_b.DT_Memory].Ca_Ear_No_Overhang_A_C[Mach_Control.Ca_b.Ca_Quantited]:=ABS(CCD.Over.Finish.AnCaOverhandX4);
	CellMemory[Mach_Control.DT_b.DT_Memory].Ca_Ear_No_Overhang_S_A[Mach_Control.Ca_b.Ca_Quantited]:=ABS(CCD.Over.Finish.PoleOverhandX4);
	
	CellMemory[Mach_Control.DT_b.DT_Memory].Ca_Ear_L_Overhang_A_C[Mach_Control.Ca_b.Ca_Quantited]:=ABS(CCD.Over.Finish.AnCaOverhandY1);
	CellMemory[Mach_Control.DT_b.DT_Memory].Ca_Ear_L_Overhang_S_A[Mach_Control.Ca_b.Ca_Quantited]:=ABS(CCD.Over.Finish.PoleOverhandY1);
	CellMemory[Mach_Control.DT_b.DT_Memory].Ca_Ear_R_Overhang_A_C[Mach_Control.Ca_b.Ca_Quantited]:=ABS(CCD.Over.Finish.AnCaOverhandY4);
	CellMemory[Mach_Control.DT_b.DT_Memory].Ca_Ear_R_Overhang_S_A[Mach_Control.Ca_b.Ca_Quantited]:=ABS(CCD.Over.Finish.PoleOverhandY4);
	
	CellMemory[Mach_Control.DT_b.DT_Memory].Ca_Cell_Overhang:=ABS(CCD.Over.Finish.AddOverhangX1);
	CellMemory[Mach_Control.DT_b.DT_Memory].Ca_Cell_Overhang_No:=ABS(CCD.Over.Finish.AddOverhangX4);
	CellMemory[Mach_Control.DT_b.DT_Memory].Ca_Cell_Overhang_L:=ABS(CCD.Over.Finish.AddOverhangY1);
	CellMemory[Mach_Control.DT_b.DT_Memory].Ca_Cell_Overhang_R:=ABS(CCD.Over.Finish.AddOverhangY4);
	
	CellMemory[Mach_Control.DT_b.DT_Memory].Ca_PoleOverhandX2[Mach_Control.Ca_b.Ca_Quantited]:=ABS(CCD.Over.Finish.PoleOverhandX2);
	CellMemory[Mach_Control.DT_b.DT_Memory].Ca_PoleOverhandX3[Mach_Control.Ca_b.Ca_Quantited]:=ABS(CCD.Over.Finish.PoleOverhandX3);
	CellMemory[Mach_Control.DT_b.DT_Memory].Ca_PoleOverhandY2[Mach_Control.Ca_b.Ca_Quantited]:=ABS(CCD.Over.Finish.PoleOverhandY2);
	CellMemory[Mach_Control.DT_b.DT_Memory].Ca_PoleOverhandY3[Mach_Control.Ca_b.Ca_Quantited]:=ABS(CCD.Over.Finish.PoleOverhandY3);
	
	CellMemory[Mach_Control.DT_b.DT_Memory].Ca_AnCaOverhandX2[Mach_Control.Ca_b.Ca_Quantited]:=ABS(CCD.Over.Finish.AnCaOverhandX2);
	CellMemory[Mach_Control.DT_b.DT_Memory].Ca_AnCaOverhandX3[Mach_Control.Ca_b.Ca_Quantited]:=ABS(CCD.Over.Finish.AnCaOverhandX3);
	CellMemory[Mach_Control.DT_b.DT_Memory].Ca_AnCaOverhandY2[Mach_Control.Ca_b.Ca_Quantited]:=ABS(CCD.Over.Finish.AnCaOverhandY2);
	CellMemory[Mach_Control.DT_b.DT_Memory].Ca_AnCaOverhandY3[Mach_Control.Ca_b.Ca_Quantited]:=ABS(CCD.Over.Finish.AnCaOverhandY3);
	
	CellMemory[Mach_Control.DT_b.DT_Memory].Ca_AddOverhangX2:=ABS(CCD.Over.Finish.AddOverhangX2);
	CellMemory[Mach_Control.DT_b.DT_Memory].Ca_AddOverhangX3:=ABS(CCD.Over.Finish.AddOverhangX3);
	CellMemory[Mach_Control.DT_b.DT_Memory].Ca_AddOverhangY2:=ABS(CCD.Over.Finish.AddOverhangY2);
	CellMemory[Mach_Control.DT_b.DT_Memory].Ca_AddOverhangY3:=ABS(CCD.Over.Finish.AddOverhangY3);
	
	CellMemory[Mach_Control.DT_b.DT_Memory].Ca_MQ_Slice[Mach_Control.Ca_b.Ca_Quantited]:=Par.stDT_date.Ca_MQ_Slice[9];
	Ca_AlarmTON[11].IN:=FALSE;
	DP_Step6:=103;	


103:
	CCD.Over.Finish.OverhandResult:=0;
	DP_Step6:=6666;	


END_CASE







CASE DP_Step7 OF
201:
	IF (CCD.Over.Finish.OverhandResult=4 OR CCD.Over.Finish.OverhandResult=2 OR CCD.Over.Finish.OverhandResult=1 ) AND NOT An_Number 
		AND ((arrAxisCtrl[AxiseNo.VirAxisName.VirMain].Status.fActPos>100 AND  arrAxisCtrl[AxiseNo.VirAxisName.VirMain].Status.fActPos<220) OR
		 (arrAxisCtrl[AxiseNo.VirAxisName.VirMain].Status.fActPos=360))THEN
		DP_Step7:=202;
	ELSIF An_Number OR Mach_Control.U.EmptyRunMode OR Mach_Control.DT_b.DT_Overhang THEN//负极报警，空跑模式，Overhang屏蔽直接跳过
		DP_Step7:=6666;	
	ELSIF   NOT An_Number AND arrAxisCtrl[AxiseNo.VirAxisName.VirMain].Status.fActPos>220 AND arrAxisCtrl[AxiseNo.VirAxisName.VirMain].Status.fActPos<360 
		AND CCD.Over.Finish.OverhandResult=0 THEN
		Mach_Control.An_b.Error[25]:=TRUE;//正极极片对齐度检测返回结果超时
		Par.stDT_date.Overhang_CSJS:=Par.stDT_date.Overhang_CSJS+1;
		DP_Step7:=6666;	
	ELSIF CCD.Over.Finish.OverhandResult=3 THEN 		
		Mach_Control.An_b.Error[27]:=TRUE; //正极极片对齐度检测返回结果无片报警
		DP_Step7:=202;	
	END_IF
							
											
202:
	CellMemory[Mach_Control.DT_b.DT_Memory].Overhang_Result[CCD.Over.Start.iPliesNo]:=CCD.Over.Finish.OverhandResult;	
	CellMemory[Mach_Control.DT_b.DT_Memory].DiaphragmUnwindingTension2[CCD.Over.Start.iPliesNo]:=LIMIT(150,ABS(Mach_Control.DT_b.DiaphragmUnwindingTension),250);
	CellMemory[Mach_Control.DT_b.DT_Memory].An_Ear_Overhang_A_C[Mach_Control.An_b.An_Quantited]:=ABS(CCD.Over.Finish.AnCaOverhandX1);
	CellMemory[Mach_Control.DT_b.DT_Memory].An_Ear_Overhang_S_CIL[Mach_Control.An_b.An_Quantited]:=ABS(CCD.Over.Finish.PoleOverhandX1);
	CellMemory[Mach_Control.DT_b.DT_Memory].An_Ear_No_Overhang_A_C[Mach_Control.An_b.An_Quantited]:=ABS(CCD.Over.Finish.AnCaOverhandX4);
	CellMemory[Mach_Control.DT_b.DT_Memory].An_Ear_No_Overhang_S_A[Mach_Control.An_b.An_Quantited]:=ABS(CCD.Over.Finish.PoleOverhandX4);
	
	CellMemory[Mach_Control.DT_b.DT_Memory].An_Ear_L_Overhang_A_C[Mach_Control.An_b.An_Quantited]:=ABS(CCD.Over.Finish.AnCaOverhandY1);
	CellMemory[Mach_Control.DT_b.DT_Memory].An_Ear_L_Overhang_S_A[Mach_Control.An_b.An_Quantited]:=ABS(CCD.Over.Finish.PoleOverhandY1);
	CellMemory[Mach_Control.DT_b.DT_Memory].An_Ear_R_Overhang_A_C[Mach_Control.An_b.An_Quantited]:=ABS(CCD.Over.Finish.AnCaOverhandY4);
	CellMemory[Mach_Control.DT_b.DT_Memory].An_Ear_R_Overhang_S_A[Mach_Control.An_b.An_Quantited]:=ABS(CCD.Over.Finish.PoleOverhandY4);
	
	CellMemory[Mach_Control.DT_b.DT_Memory].An_Cell_Overhang:=ABS(CCD.Over.Finish.AddOverhangX1);
	CellMemory[Mach_Control.DT_b.DT_Memory].An_Cell_Overhang_No:=ABS(CCD.Over.Finish.AddOverhangX4);
	CellMemory[Mach_Control.DT_b.DT_Memory].An_Cell_Overhang_L:=ABS(CCD.Over.Finish.AddOverhangY1);
	CellMemory[Mach_Control.DT_b.DT_Memory].An_Cell_Overhang_R:=ABS(CCD.Over.Finish.AddOverhangY4);
	
	CellMemory[Mach_Control.DT_b.DT_Memory].An_PoleOverhandX2[Mach_Control.An_b.An_Quantited]:=ABS(CCD.Over.Finish.PoleOverhandX2);
	CellMemory[Mach_Control.DT_b.DT_Memory].An_PoleOverhandX3[Mach_Control.An_b.An_Quantited]:=ABS(CCD.Over.Finish.PoleOverhandX3);
	CellMemory[Mach_Control.DT_b.DT_Memory].An_PoleOverhandY2[Mach_Control.An_b.An_Quantited]:=ABS(CCD.Over.Finish.PoleOverhandY2);
	CellMemory[Mach_Control.DT_b.DT_Memory].An_PoleOverhandY3[Mach_Control.An_b.An_Quantited]:=ABS(CCD.Over.Finish.PoleOverhandY3);
	
	CellMemory[Mach_Control.DT_b.DT_Memory].An_AnCaOverhandX2[Mach_Control.An_b.An_Quantited]:=ABS(CCD.Over.Finish.AnCaOverhandX2);
	CellMemory[Mach_Control.DT_b.DT_Memory].An_AnCaOverhandX3[Mach_Control.An_b.An_Quantited]:=ABS(CCD.Over.Finish.AnCaOverhandX3);
	CellMemory[Mach_Control.DT_b.DT_Memory].An_AnCaOverhandY2[Mach_Control.An_b.An_Quantited]:=ABS(CCD.Over.Finish.AnCaOverhandY2);
	CellMemory[Mach_Control.DT_b.DT_Memory].An_AnCaOverhandY3[Mach_Control.An_b.An_Quantited]:=ABS(CCD.Over.Finish.AnCaOverhandY3);
	
	CellMemory[Mach_Control.DT_b.DT_Memory].An_AddOverhangX2:=ABS(CCD.Over.Finish.AddOverhangX2);
	CellMemory[Mach_Control.DT_b.DT_Memory].An_AddOverhangX3:=ABS(CCD.Over.Finish.AddOverhangX3);
	CellMemory[Mach_Control.DT_b.DT_Memory].An_AddOverhangY2:=ABS(CCD.Over.Finish.AddOverhangY2);
	CellMemory[Mach_Control.DT_b.DT_Memory].An_AddOverhangY3:=ABS(CCD.Over.Finish.AddOverhangY3);
	
	CellMemory[Mach_Control.DT_b.DT_Memory].An_MQ_Slice[Mach_Control.An_b.An_Quantited]:=Par.stDT_date.An_MQ_Slice[2];
	DP_Step7:=203;	

203:
	CCD.Over.Finish.OverhandResult:=0;
	DP_Step7:=6666;

END_CASE



CASE DP_Step8 OF	
100:
	Ca_StandbySub3_ton[2].IN:=FALSE;
	IF  NOT Mach_Control.U.CCD_ChosesHMI  AND NOT  Mach_Control.U.EmptyRunMode  THEN
		//IF arrAxis[AxiseNo.VirAxisName.VirMain].NcToPlc.SetPos>109 AND arrAxis[AxiseNo.VirAxisName.VirMain].NcToPlc.SetPos<=112   THEN
		IF arrAxis[AxiseNo.VirAxisName.VirMain].NcToPlc.SetPos>110 AND arrAxis[AxiseNo.VirAxisName.VirMain].NcToPlc.SetPos<=115   THEN
				CCD.CaRec.Finish.RectifyX1:=0;
				CCD.CaRec.Finish.RectifyX2:=0;
				CCD.CaRec.Finish.RectifyY:=0;		
				CCD.CaRec.Finish.RectifyResult:=0;//拍照结果清零									
				Mach_Control.Ca_b.Ca_CCDStart :=TRUE;//启动CCD拍照
				CCD.CaRec.Start.iPhotoDo:=1;//启动CCD第二次拍照
				//arrCyCtrl[arrCyNo.ElectValveName.CadeviationIonizedWind].Cmd.bON:=TRUE;//负极纠偏平台除尘
				//arrCyCtrl[arrCyNo.ElectValveName.AndeviationIonizedWind].Cmd.bON:=TRUE;//正极纠偏平台除尘
				DP_Step8:=110;
		END_IF
	ELSE
		DP_Step8:=6661;
	END_IF
110:
	Ca_StandbySub3_ton[2].IN:=CCD.CaRec.Finish.RectifyResult=0;
	IF Ca_StandbySub3_ton[2].Q THEN
		Mach_Control.DT_b.Error[51]:=TRUE;//检测负极纠偏平台空片结果返回超时
		DP_Step8:=9991;
	ELSIF CCD.CaRec.Finish.RectifyResult<>0 AND CCD.CaRec.Finish.RectifyResult<>3   THEN
		Mach_Control.Ca_b.Error[24]:=TRUE;//负极纠偏平台NG片未排掉报警，请拿掉
		Ca_StandbySub3_ton[2].IN:=FALSE;
		DP_Step8:=9992;
	ELSIF CCD.CaRec.Finish.RectifyResult=3  THEN
		DP_Step8:=6661;
	END_IF

200:
	An_StandbySub3_ton[2].IN:=FALSE;
	IF  NOT Mach_Control.U.CCD_ChosesHMI  AND NOT  Mach_Control.U.EmptyRunMode    THEN
		//IF arrAxis[AxiseNo.VirAxisName.VirMain].NcToPlc.SetPos>118 AND arrAxis[AxiseNo.VirAxisName.VirMain].NcToPlc.SetPos<=123  THEN
		IF arrAxis[AxiseNo.VirAxisName.VirMain].NcToPlc.SetPos>110 AND arrAxis[AxiseNo.VirAxisName.VirMain].NcToPlc.SetPos<=115   THEN
			CCD.AnRec.Finish.RectifyResult:=0;
			CCD.AnRec.Finish.RectifyX1:=0;
			CCD.AnRec.Finish.RectifyX2:=0;
			CCD.AnRec.Finish.RectifyY:=0;												
			Mach_Control.An_b.An_CCDStart :=TRUE;//启动CCD拍照
			CCD.AnRec.Start.iPhotoDo:=1;//第二次拍照
			//arrCyCtrl[arrCyNo.ElectValveName.CadeviationIonizedWind].Cmd.bON:=TRUE;//负极纠偏平台除尘
			//arrCyCtrl[arrCyNo.ElectValveName.AndeviationIonizedWind].Cmd.bON:=TRUE;//正极纠偏平台除尘
			DP_Step8:=210;
		END_IF
	ELSE
		DP_Step8:=6662;
	END_IF	
210:
	An_StandbySub3_ton[2].IN:=CCD.AnRec.Finish.RectifyResult=0;
	IF An_StandbySub3_ton[2].Q THEN				
		Mach_Control.DT_b.Error[52]:=TRUE;//检测正极纠偏平台空片结果返回超时
		An_StandbySub3_ton[2].IN:=FALSE;
		DP_Step8:=9993;		
	ELSIF CCD.AnRec.Finish.RectifyResult<>0 AND CCD.AnRec.Finish.RectifyResult<>3 THEN
		Mach_Control.An_b.Error[24]:=TRUE;//正极纠偏平台NG片未排掉报警，请拿掉 
		An_StandbySub3_ton[2].IN:=FALSE;
		DP_Step8:=9994;
	ELSIF CCD.AnRec.Finish.RectifyResult=3 THEN
		An_StandbySub3_ton[2].IN:=FALSE;
		DP_Step8:=6662;
	END_IF
	
END_CASE

*)
END_ACTION

ACTION _01DT_Auto3:

(*******************************************************************************************************叠完片后，空叠片隔膜***************************************************************************************************************************)
DT_TON[5](IN:= , PT:=T#300MS , Q=> , ET=> );//

IF Mach_Control.U.DT_iMode=1 THEN//在自动状态下
CASE DP_Step0 OF    //空叠隔膜流程
1000://判断主轴是否停止、是否在初始位、是否有轴在耦合中
	IF NOT DP_SinStepe THEN
		IF arrAxisCtrl[AxiseNo.VirAxisName.VirMain].Status.NoMoving AND arrAxisCtrl[AxiseNo.VirAxisName.VirMain].Status.fSetPos=0 AND NOT DT_AxiseCoupling THEN
			KD_Mark:=TRUE;//空叠隔膜中
			IF Mach_Control.DT_b.SinStepMode THEN//单步调试模式
				DP_SinStepe:=TRUE;
			ELSE
				DP_SinStepe:=FALSE;	
			END_IF
			DP_Step0:=1020;
		ELSE
			DP_Step1:=100;//解除耦合，主轴回零
			DP_Step0:=1010;
		END_IF
	END_IF
1010://判断主轴当前的当前位置是否为0
	IF DP_Step1=6666 AND arrAxisCtrl[AxiseNo.VirAxisName.VirMain].Status.NoMoving AND arrAxisCtrl[AxiseNo.VirAxisName.VirMain].Status.fSetPos=0 AND NOT DT_AxiseCoupling THEN
		IF Mach_Control.DT_b.SinStepMode THEN//单步调试模式
			DP_SinStepe:=TRUE;
		ELSE
			DP_SinStepe:=FALSE;	
		END_IF									
		DP_Step0:=1020;
	END_IF	

1020://判断NG气缸是否在安全位
	IF arrCyCtrl[arrCyNo.CylinderName.AnScrapbinCy].Status.ONState AND arrCyCtrl[arrCyNo.CylinderName.CaScrapbinUDCy].Status.OFFState AND
		arrCyCtrl[arrCyNo.CylinderName.CaScrapbinCy].Status.ONState AND arrCyCtrl[arrCyNo.CylinderName.PreDiaph].Status.OFFState AND 
		arrCyCtrl[arrCyNo.CylinderName.PoleHotCutterCy].Status.OFFState AND arrCyCtrl[arrCyNo.CylinderName.PoleTapeCy].Status.OFFState AND
		arrCyCtrl[arrCyNo.CylinderName.PoleTapeSplicerRCy].Status.ONState AND arrCyCtrl[arrCyNo.CylinderName.PoleTapeSplicerLCy].Status.ONState THEN
		DP_Step0:=1050;		
	ELSE
		DP_Step0:=1030;	
	END_IF
1030:
	arrCyCtrl[arrCyNo.CylinderName.AnScrapbinCy].Cmd.bON:=TRUE;
	arrCyCtrl[arrCyNo.CylinderName.PreDiaph].Cmd.bOFF:=TRUE;
	arrCyCtrl[arrCyNo.CylinderName.PoleHotCutterCy].Cmd.bOFF:=TRUE;
	arrCyCtrl[arrCyNo.CylinderName.PoleTapeCy].Cmd.bOFF:=TRUE;
	arrCyCtrl[arrCyNo.CylinderName.PoleTapeSplicerRCy].Cmd.bON:=TRUE;
	arrCyCtrl[arrCyNo.CylinderName.PoleTapeSplicerLCy].Cmd.bON:=TRUE;
	arrCyCtrl[arrCyNo.CylinderName.CaScrapbinCy].Cmd.bON:=TRUE;
	IF   arrCyCtrl[arrCyNo.CylinderName.AnScrapbinCy].Status.ONState AND  arrCyCtrl[arrCyNo.CylinderName.PreDiaph].Status.OFFState AND 
	arrCyCtrl[arrCyNo.CylinderName.PoleHotCutterCy].Status.OFFState AND arrCyCtrl[arrCyNo.CylinderName.PoleTapeCy].Status.OFFState AND
	arrCyCtrl[arrCyNo.CylinderName.PoleTapeSplicerRCy].Status.ONState AND arrCyCtrl[arrCyNo.CylinderName.PoleTapeSplicerLCy].Status.ONState
	AND arrCyCtrl[arrCyNo.CylinderName.CaScrapbinCy].Cmd.bON THEN
		DP_Step0:=1040;									
	END_IF
1040:
	arrCyCtrl[arrCyNo.CylinderName.CaScrapbinUDCy].Cmd.bOFF:=TRUE;
	IF  arrCyCtrl[arrCyNo.CylinderName.CaScrapbinUDCy].Status.OFFState THEN
		DP_Step0:=1050;	
	END_IF						
1050://	最后一层为负极片，所以，最开始先叠正极的隔膜
	KD_Mark:=TRUE;//空叠隔膜中
	IF NOT Bnt_Blueflaging THEN
		IF Mach_Control.An_b.An_KDQuantited  = Mach_Control.Ca_b.Ca_KDQuantited   THEN//先叠正极
			DP_Step0:=1100;
		ELSIF Mach_Control.An_b.An_KDQuantited  > Mach_Control.Ca_b.Ca_KDQuantited   THEN//先叠负极
			DP_Step0:=1500;
		END_IF
	ELSE//判断隔膜平移轴位置
		IF AN_CarryingPos1 THEN	
			DP_Step0:=1100;			
		ELSIF Ca_CarryingPos1 THEN
			DP_Step0:=1500;	
		ELSE
			Mach_Control.DT_b.Error[57]:=TRUE;//空叠隔膜时正负极都不在取片位	
		END_IF	
	(*
		IF (Mach_Control.An_b.An_KDQuantited  <= Mach_Control.Ca_b.Ca_KDQuantited) AND AN_CarryingPos1   THEN//先叠正极
			DP_Step0:=1100;
		ELSE 
			IF Ca_CarryingPos1 THEN	
				DP_Step0:=1500;	
			ELSE
				;//空叠隔膜时正负极都不在取片位	
			END_IF
		END_IF
	*)
	END_IF		

1100://判断叠台搬运机械手是否有片
	IF AN_CarryingPos1  THEN//正极搬运、叠片各轴在初始位	
		IF arrCyCtrl[arrCyNo.ElectValveName.AnDTCarryingVacuum].Io.DIOnSwitch AND  Mach_Control.An_b.An_DPCarryingFalg THEN//正极再取片位且叠台搬运有片,把当前片放到纠偏台
			DP_Step0:=1150;
		ELSE
			DP_Step0:=2000;	
		END_IF
	ELSE
		Mach_Control.DT_b.Error[8]:=TRUE;//叠正极片凸轮耦合时，正极片不在取片位
		DP_Step0:=10001;
	END_IF	
	
1150://纠偏台回初始位
	//纠偏平台X1移动至初始位
	IF NOT DP_SinStepe THEN
		IF arrAxisCtrl[AxiseNo.AxisName.AndeviationX1].Status.Homed  AND arrAxisCtrl[AxiseNo.AxisName.AndeviationX1].Status.NoMoving AND NOT  arrAxisCtrl[AxiseNo.AxisName.AndeviationX1].Status.Error THEN
			IF arrAxisCtrl[AxiseNo.AxisName.AndeviationX1].Cmd.arrbRealPoint[1] THEN
				arrAxisCtrl[AxiseNo.AxisName.AndeviationX1].Cmd.iGoSetPos:=0;
			ELSE
				arrAxisCtrl[AxiseNo.AxisName.AndeviationX1].Cmd.iGoSetPos:=1;
			END_IF					
		END_IF
		//纠偏平台X2移动至初始位
		IF arrAxisCtrl[AxiseNo.AxisName.AndeviationX2].Status.Homed  AND arrAxisCtrl[AxiseNo.AxisName.AndeviationX2].Status.NoMoving AND NOT  arrAxisCtrl[AxiseNo.AxisName.AndeviationX2].Status.Error THEN
			IF arrAxisCtrl[AxiseNo.AxisName.AndeviationX2].Cmd.arrbRealPoint[1] THEN
				arrAxisCtrl[AxiseNo.AxisName.AndeviationX2].Cmd.iGoSetPos:=0;
			ELSE
				arrAxisCtrl[AxiseNo.AxisName.AndeviationX2].Cmd.iGoSetPos:=1;
			END_IF					
		END_IF
		//纠偏平台X2移动至初始位
		IF arrAxisCtrl[AxiseNo.AxisName.AndeviationY].Status.Homed  AND arrAxisCtrl[AxiseNo.AxisName.AndeviationY].Status.NoMoving AND NOT  arrAxisCtrl[AxiseNo.AxisName.AndeviationY].Status.Error THEN
			IF arrAxisCtrl[AxiseNo.AxisName.AndeviationY].Cmd.arrbRealPoint[1] THEN
				arrAxisCtrl[AxiseNo.AxisName.AndeviationY].Cmd.iGoSetPos:=0;
			ELSE
				arrAxisCtrl[AxiseNo.AxisName.AndeviationY].Cmd.iGoSetPos:=1;
			END_IF					
		END_IF
		IF arrAxisCtrl[AxiseNo.AxisName.AndeviationX1].Cmd.arrbRealPoint[1] AND arrAxisCtrl[AxiseNo.AxisName.AndeviationX2].Cmd.arrbRealPoint[1] AND arrAxisCtrl[AxiseNo.AxisName.AndeviationY].Cmd.arrbRealPoint[1] THEN
			DT_SingeMode();//单步选择	
			DP_Step0:=1200;	
			DT_TON[5].IN:=FALSE;
		END_IF	
	END_IF
1200:
	IF NOT DP_SinStepe THEN
		IF arrAxisCtrl[AxiseNo.AxisName.AnDTCarryingUpDown].Cmd.arrbRealPoint[3] THEN
			arrAxisCtrl[AxiseNo.AxisName.AnDTCarryingUpDown].Cmd.iGoSetPos:=0;
			/// 吸盘破真空    纠偏台开真空
			arrCyCtrl[arrCyNo.ElectValveName.AnDTCarryingVacuum].Cmd.bON:=TRUE;	//正极叠台搬运升降真空	真空
			arrCyCtrl[arrCyNo.ElectValveName.AnDTCarryingVacuum].Cmd.bOFF:=FALSE;	//正极叠台搬运升降真空破真空		
			arrCyCtrl[arrCyNo.ElectValveName.AnDTCarryingVacuumBark].Cmd.bON:=TRUE;	//正极叠台搬运升降真空	真空
			arrCyCtrl[arrCyNo.ElectValveName.AnDTCarryingVacuumBark].Cmd.bOFF:=FALSE;	//正极叠台搬运升降真空破真空											
			arrCyCtrl[arrCyNo.ElectValveName.AndeviationVacuum].Cmd.bON:=TRUE;	//正极纠偏台真空			
			arrCyCtrl[arrCyNo.ElectValveName.AndeviationVacuum].Cmd.bOFF:=FALSE;	//正极纠偏台真空	
			DT_SingeMode();//单步选择	
			DP_Step0:=1250;
			DT_TON[5].IN:=TRUE;
		ELSE
			arrAxisCtrl[AxiseNo.AxisName.AnDTCarryingUpDown].Cmd.iGoSetPos:=3;//负极搬运升降2上升至凸轮耦合初始高度
		END_IF	
	END_IF	
1250://叠台搬运极片放回纠偏台
	IF NOT DP_SinStepe THEN
		  IF DT_TON[5].Q THEN
				IF arrAxisCtrl[AxiseNo.AxisName.AnDTCarryingUpDown].Cmd.arrbRealPoint[4] THEN
					arrAxisCtrl[AxiseNo.AxisName.AnDTCarryingUpDown].Cmd.iGoSetPos:=0;
					/// 吸盘破真空    纠偏台开真空
					Mach_Control.An_b.An_deviationFalg:=TRUE;//复位纠偏平台有料标记
					Mach_Control.An_b.An_DPCarryingFalg:=FALSE;//负极搬运真空吸盘有料标记复位
					Par.stDT_date.An_MQ_Slice[1]:=Par.stDT_date.An_MQ_Slice[2];
					DT_SingeMode();//单步选择	
					DP_Step0:=1300;
					DT_TON[5].IN:=FALSE;
				ELSE
					arrAxisCtrl[AxiseNo.AxisName.AnDTCarryingUpDown].Cmd.iGoSetPos:=4;//负极搬运升降2上升至凸轮耦合初始高度
				END_IF	
		 END_IF		
	END_IF			
1300:
	DP_Step0:=2000;	
	

	
	
	
1500://判断负极叠台搬运是否有片，有片的话放到纠偏台
	IF NOT DP_SinStepe THEN
		IF CA_CarryingPos1  THEN//负极搬运、叠片各轴在初始位
			IF arrCyCtrl[arrCyNo.ElectValveName.CaDTCarryingVacuum].Io.DIOnSwitch AND  Mach_Control.Ca_b.Ca_DPCarryingFalg THEN//正极再取片位且叠台搬运有片,把当前片放到纠偏台
				DP_Step0:=1550;
			ELSE
				DP_Step0:=3000;	
			END_IF
		ELSE
			IF (Ca_Step0=0 OR Ca_Step0=6666) AND (Ca_Step3=0 OR Ca_Step3=6666) AND Scan_TON[2].Q THEN
				Scan_TON[2].IN:=FALSE;		
				DP_Step0:=9994;
				DTPosError[2]:=TRUE;
			END_IF
		END_IF
	END_IF	
1550://纠偏台回初始位
	//纠偏平台X1移动至初始位
	IF NOT DP_SinStepe THEN
		IF arrAxisCtrl[AxiseNo.AxisName.CadeviationX1].Status.Homed  AND arrAxisCtrl[AxiseNo.AxisName.CadeviationX1].Status.NoMoving AND NOT  arrAxisCtrl[AxiseNo.AxisName.CadeviationX1].Status.Error THEN
			IF arrAxisCtrl[AxiseNo.AxisName.CadeviationX1].Cmd.arrbRealPoint[1] THEN
				arrAxisCtrl[AxiseNo.AxisName.CadeviationX1].Cmd.iGoSetPos:=0;
			ELSE
				arrAxisCtrl[AxiseNo.AxisName.CadeviationX1].Cmd.iGoSetPos:=1;
			END_IF					
		END_IF
		//纠偏平台X2移动至初始位
		IF arrAxisCtrl[AxiseNo.AxisName.CadeviationX2].Status.Homed  AND arrAxisCtrl[AxiseNo.AxisName.CadeviationX2].Status.NoMoving AND NOT  arrAxisCtrl[AxiseNo.AxisName.CadeviationX2].Status.Error THEN
			IF arrAxisCtrl[AxiseNo.AxisName.CadeviationX2].Cmd.arrbRealPoint[1] THEN
				arrAxisCtrl[AxiseNo.AxisName.CadeviationX2].Cmd.iGoSetPos:=0;
			ELSE
				arrAxisCtrl[AxiseNo.AxisName.CadeviationX2].Cmd.iGoSetPos:=1;
			END_IF					
		END_IF
		//纠偏平台X2移动至初始位
		IF arrAxisCtrl[AxiseNo.AxisName.CadeviationY].Status.Homed  AND arrAxisCtrl[AxiseNo.AxisName.CadeviationY].Status.NoMoving AND NOT  arrAxisCtrl[AxiseNo.AxisName.CadeviationY].Status.Error THEN
			IF arrAxisCtrl[AxiseNo.AxisName.CadeviationY].Cmd.arrbRealPoint[1] THEN
				arrAxisCtrl[AxiseNo.AxisName.CadeviationY].Cmd.iGoSetPos:=0;
			ELSE
				arrAxisCtrl[AxiseNo.AxisName.CadeviationY].Cmd.iGoSetPos:=1;
			END_IF					
		END_IF
		IF arrAxisCtrl[AxiseNo.AxisName.CadeviationX1].Cmd.arrbRealPoint[1] AND arrAxisCtrl[AxiseNo.AxisName.CadeviationX2].Cmd.arrbRealPoint[1] AND arrAxisCtrl[AxiseNo.AxisName.CadeviationY].Cmd.arrbRealPoint[1] THEN
			DT_SingeMode();//单步选择	
			DP_Step0:=1600;	
			DT_TON[5].IN:=FALSE;
		END_IF	
	END_IF
1600:
	IF NOT DP_SinStepe THEN
		IF arrAxisCtrl[AxiseNo.AxisName.CaDTCarryingUpDown].Cmd.arrbRealPoint[3] THEN
			arrAxisCtrl[AxiseNo.AxisName.CaDTCarryingUpDown].Cmd.iGoSetPos:=0;
			/// 吸盘破真空    纠偏台开真空
			arrCyCtrl[arrCyNo.ElectValveName.CaDTCarryingVacuum].Cmd.bON:=TRUE;	//负极叠台搬运升降真空	真空
			arrCyCtrl[arrCyNo.ElectValveName.CaDTCarryingVacuum].Cmd.bOFF:=FALSE;	//负极叠台搬运升降真空破真空								
			arrCyCtrl[arrCyNo.ElectValveName.CadeviationVacuum].Cmd.bON:=TRUE;	//负极纠偏台真空			
			arrCyCtrl[arrCyNo.ElectValveName.CadeviationVacuum].Cmd.bOFF:=FALSE;	//负极纠偏台真空	   
			DT_SingeMode();//单步选择	
			DP_Step0:=1650;
			DT_TON[5].IN:=TRUE;
		ELSE
			arrAxisCtrl[AxiseNo.AxisName.CaDTCarryingUpDown].Cmd.iGoSetPos:=3;//负极搬运升降2上升至凸轮耦合初始高度
		END_IF	
	END_IF
1650://叠台搬运极片放回纠偏台
	IF NOT DP_SinStepe THEN
		 IF DT_TON[5].Q THEN
				IF arrAxisCtrl[AxiseNo.AxisName.CaDTCarryingUpDown].Cmd.arrbRealPoint[4] THEN
					arrAxisCtrl[AxiseNo.AxisName.CaDTCarryingUpDown].Cmd.iGoSetPos:=0;
					/// 吸盘破真空    纠偏台开真空
					Mach_Control.Ca_b.Ca_deviationFalg:=TRUE;//复位纠偏平台有料标记
					Mach_Control.Ca_b.Ca_DPCarryingFalg:=FALSE;//负极搬运真空吸盘有料标记复位
					Par.stDT_date.Ca_MQ_Slice[8]:=Par.stDT_date.Ca_MQ_Slice[9];
					DT_SingeMode();//单步选择	
					DP_Step0:=1700;
					DT_TON[5].IN:=FALSE;
				ELSE
					arrAxisCtrl[AxiseNo.AxisName.CaDTCarryingUpDown].Cmd.iGoSetPos:=4;//负极搬运升降2上升至凸轮耦合初始高度
				END_IF		
	    END_IF	
	END_IF	
1700:
	DP_Step0:=3000;	
	


	
2000:		
	IF NOT DP_SinStepe THEN
		IF AN_CarryingPos1  THEN//正极搬运、叠片各轴在初始位										
			IF CA_CarryingPos2 THEN//负极在叠片位
				IF arrAxisCtrl[AxiseNo.AxisName.SEPTATLine].Cmd.arrbRealPoint[1]  THEN
					IF Mach_Control.DT_b.SinStepMode THEN//单步调试模式
						DP_SinStepe:=TRUE;
					ELSE
						DP_SinStepe:=FALSE;	
					END_IF
					DP_Step0:=2010;//
				ELSE
					Mach_Control.DT_b.Error[6]:=TRUE;//叠正极片凸轮耦合时，隔膜平移轴即不在负极叠片位，也不在正极叠片位报警
					DP_Step0:=9998;
				END_IF;
			ELSIF  CA_CarryingPos1  THEN //负极取片位
				IF arrAxisCtrl[AxiseNo.AxisName.SEPTATLine].Cmd.arrbRealPoint[1]  THEN
					IF Mach_Control.DT_b.SinStepMode THEN//单步调试模式
						DP_SinStepe:=TRUE;
					ELSE
						DP_SinStepe:=FALSE;	
					END_IF
					DP_Step0:=2030;//
				ELSIF arrAxisCtrl[AxiseNo.AxisName.SEPTATLine].Cmd.arrbRealPoint[2]  THEN
					IF Mach_Control.DT_b.SinStepMode THEN//单步调试模式
						DP_SinStepe:=TRUE;
					ELSE
						DP_SinStepe:=FALSE;	
					END_IF
					DP_Step0:=2050;//
				ELSE
					Mach_Control.DT_b.Error[6]:=TRUE;//叠正极片凸轮耦合时，隔膜平移轴即不在负极叠片位，也不在正极叠片位报警
					DP_Step0:=9999;
				END_IF;							
			ELSE
				Mach_Control.DT_b.Error[7]:=TRUE;//叠正极片凸轮耦合时，负极取片即不在取片位，也不在叠片位
				DP_Step0:=10000;
			END_IF
		ELSE
			Mach_Control.DT_b.Error[8]:=TRUE;//叠正极片凸轮耦合时，正极片不在取片位
			DP_Step0:=10001;
		END_IF
	END_IF		


2010://负极搬运、叠片各轴在初始位，隔膜平移轴负极叠片位、正极叠片在放极片初始位
	IF NOT DP_SinStepe THEN
		An_CanIn5:=TRUE;
		IF Mach_Control.DT_b.SinStepMode THEN//单步调试模式
				DP_SinStepe:=TRUE;
			ELSE
				DP_SinStepe:=FALSE;	
			END_IF
		DP_Step0:=2020;	
	END_IF	
2020:
	IF NOT DP_SinStepe THEN
		IF NOT An_CanIn5 THEN
			IF Mach_Control.DT_b.SinStepMode THEN//单步调试模式
				DP_SinStepe:=TRUE;
			ELSE
				DP_SinStepe:=FALSE;	
			END_IF	
			DP_Step0:=2070;
		ELSIF fbAnCamInCarryingLine.bError  OR fbAnCamInDTCarryingLine.bError OR fbAnCamInDTCarryingUpDown.bError OR 
			fbAnCamInCarryingWhirling.bError OR fbCaCamInCarryingLine2.bError OR 
			fbCaCamInDTCarryingUpDown.bError OR fbCamInGMBuffer.bError OR fbCamInGMDanserMove.bError OR fbCamInVirGMDriver.bError   OR
			fbCamInRightYDUpDown.bError OR fbCamInRightYDLine.bError  THEN
			An_CanIn5:=FALSE;
			Mach_Control.DT_b.Error[19]:=TRUE;//凸轮耦合报警
			DP_Step0:=10004;		
		END_IF
	END_IF		
2030://负极搬运、叠片各轴在初始位，隔膜平移轴负极叠片位、正极叠片在取极片位
	IF NOT DP_SinStepe THEN
		IF Mach_Control.DT_b.SinStepMode THEN//单步调试模式
			DP_SinStepe:=TRUE;
		ELSE
			DP_SinStepe:=FALSE;	
		END_IF
		An_CanIn6:=TRUE;
		DP_Step0:=2040;
	END_IF
2040:
	IF NOT DP_SinStepe THEN
		IF NOT An_CanIn6 THEN
			IF Mach_Control.DT_b.SinStepMode THEN//单步调试模式
				DP_SinStepe:=TRUE;
			ELSE
				DP_SinStepe:=FALSE;	
			END_IF
			DP_Step0:=2070;
		ELSIF fbAnCamInCarryingLine.bError OR fbAnCamInDTCarryingLine.bError OR
			fbAnCamInDTCarryingUpDown.bError OR fbAnCamInCarryingWhirling.bError OR fbCamInGMBuffer.bError OR
			fbCamInGMDanserMove.bError OR fbCamInVirGMDriver.bError  OR fbCamInRightYDUpDown.bError OR
			fbCamInRightYDLine.bError  THEN
			An_CanIn6:=FALSE;
			Mach_Control.DT_b.Error[19]:=TRUE;//凸轮耦合报警
			DP_Step0:=10002;									
		END_IF
	END_IF
2050://负极搬运、叠片各轴在初始位，隔膜平移轴正极叠片位、正极叠片在取极片位
	IF NOT DP_SinStepe THEN
		An_CanIn7:=TRUE;
		IF Mach_Control.DT_b.SinStepMode THEN//单步调试模式
				DP_SinStepe:=TRUE;
			ELSE
				DP_SinStepe:=FALSE;	
			END_IF
		DP_Step0:=2060;
	END_IF
2060:
	IF NOT DP_SinStepe THEN
			arrAxisCtrl[AxiseNo.VirAxisName.VirMain].Cmd	.bMoveAbs:=FALSE;	
			IF NOT An_CanIn7 THEN
				IF Mach_Control.DT_b.SinStepMode THEN//单步调试模式
					DP_SinStepe:=TRUE;
				ELSE
					DP_SinStepe:=FALSE;	
				END_IF
				DP_Step0:=2070;
			ELSIF fbAnCamInCarryingLine.bError OR fbAnCamInCarryingUpDown.bError OR fbAnCamInDTCarryingLine.bError OR fbAnCamInDTCarryingUpDown.bError OR 
				fbAnCamInCarryingWhirling.bError OR fbCamInRightYDUpDown.bError OR fbCamInRightYDLine.bError THEN
				An_CanIn7:=FALSE;
				Mach_Control.DT_b.Error[19]:=TRUE;//凸轮耦合报警
				DP_Step0:=10003;												
			END_IF
	END_IF	
	
2070://判断正极叠片搬运机械手上是否有极片

	IF NOT DP_SinStepe THEN
		VirMain_TON.IN:=FALSE;
		IF (NOT arrCyCtrl[arrCyNo.ElectValveName.AnDTCarryingVacuum].Io.DIOnSwitch AND NOT Mach_Control.An_b.An_DPCarryingFalg) OR Bnt_Blueflaging THEN	
			IF Mach_Control.DT_b.SinStepMode THEN//单步调试模式
				DP_SinStepe:=TRUE;
			ELSE
				DP_SinStepe:=FALSE;	
			END_IF
			DP_Step0:=2071;
		ELSE	
		  	Mach_Control.An_b.Error[28]:=TRUE; //正极叠片完空叠隔膜时，正极叠片搬运机械手真空有信号、标记有极片报警,请拿掉极片
		END_IF  
	END_IF

2071://主轴启动
	IF NOT DP_SinStepe THEN
		arrAxisCtrl[AxiseNo.VirAxisName.VirMain].Cmd	.bDynamitcsParSel:=2;	
		arrAxisPar[AxiseNo.VirAxisName.VirMain].fTagatTime:=VirMain_TagatTime;
		arrAxisCtrl[AxiseNo.VirAxisName.VirMain].Cmd	.fPositon_of_Abs:=360;
		arrAxisCtrl[AxiseNo.VirAxisName.VirMain].Cmd	.bMoveAbs:=TRUE;	
		//fbCaCamInCarryingUpDown2OutCamFlge:=FALSE;//负极升降2凸轮解耦标记										
		IF  arrAxis[AxiseNo.VirAxisName.VirMain].Status.Moving OR arrAxisCtrl[AxiseNo.VirAxisName.VirMain].Status.fActPos>=10  THEN
			VirMain_TON.IN:=FALSE;
			arrAxisCtrl[AxiseNo.VirAxisName.VirMain].Cmd	.bMoveAbs:=FALSE;	
			DP_Step0:=2080;	
		ELSE
			IF NOT VirMain_TON.Q THEN
				VirMain_TON.IN:=TRUE;
			ELSE
				VirMain_TON.IN:=FALSE;
				Mach_Control.DT_b.Error[22]:=TRUE;//主轴启动超时报警
				DP_Step0:=10006;	
			END_IF	
		END_IF	
	END_IF				
			
(*2080:
IF arrAxis[AxiseNo.VirAxisName.VirMain].NcToPlc.SetPos>=234 AND arrAxis[AxiseNo.VirAxisName.VirMain].NcToPlc.SetPos<=240 THEN
	arrCyCtrl[arrCyNo.ElectValveName.AnDTCarryingVacuum].Cmd.bOFF:=TRUE;//正极叠片搬运真空关
	arrCyCtrl[arrCyNo.ElectValveName.AnDTCarryingVacuumBark].Cmd.bON:=TRUE;//正极叠片搬运破真空开
	Mach_Control.An_b.An_DPCarryingFalg :=FALSE;//复位正极叠片搬运吸盘上有料标记																									
END_IF				
IF arrAxis[AxiseNo.VirAxisName.VirMain].NcToPlc.SetPos=360 AND  arrAxis[AxiseNo.VirAxisName.VirMain].Status.NotMoving  THEN
			Mach_Control.An_b.An_KDQuantited:=Mach_Control.An_b.An_KDQuantited +1;
			DP_Step1:=100;//解除耦合，主轴回零子程序
			arrAxisCtrl[AxiseNo.AxisName.DTUpDown].Cmd.fPosition_of_Rel:=-Par.stDT_date.SEPTA_Thickness;
			arrAxisPar[AxiseNo.AxisName.DTUpDown].fVelocity_of_Rel:=100;
			arrAxisCtrl[AxiseNo.AxisName.DTUpDown].Cmd.bMoveRel:=TRUE;
			DP_Step0:=0;
END_IF*)

3000:
	IF NOT DP_SinStepe THEN		
		Scan_TON[2].IN:=TRUE;	
		IF CA_CarryingPos1  THEN//负极搬运、叠片各轴在初始位
			Scan_TON[1].IN:=TRUE;	
			IF AN_CarryingPos2  THEN//正极在叠片位	
				IF arrAxisCtrl[AxiseNo.AxisName.SEPTATLine].Cmd.arrbRealPoint[2]   THEN													
					IF Mach_Control.DT_b.SinStepMode THEN//单步调试模式
						DP_SinStepe:=TRUE;
					ELSE
						DP_SinStepe:=FALSE;	
					END_IF												
					DP_Step0:=3010;//													
				ELSE
					Mach_Control.DT_b.Error[5]:=TRUE;//叠负极片凸轮耦合时，隔膜平移轴即不在负极叠片位，也不在正极叠片位报警
					DP_Step0:=9991;	
				END_IF;
			ELSIF AN_CarryingPos1  THEN//在取片位																		
				IF arrAxisCtrl[AxiseNo.AxisName.SEPTATLine].Cmd.arrbRealPoint[1]  THEN
					IF Mach_Control.DT_b.SinStepMode THEN//单步调试模式
						DP_SinStepe:=TRUE;
					ELSE
						DP_SinStepe:=FALSE;	
					END_IF											
					DP_Step0:=3030;//
				ELSIF arrAxisCtrl[AxiseNo.AxisName.SEPTATLine].Cmd.arrbRealPoint[2] THEN
					IF Mach_Control.DT_b.SinStepMode THEN//单步调试模式
						DP_SinStepe:=TRUE;
					ELSE
						DP_SinStepe:=FALSE;	
					END_IF											
					DP_Step0:=3050;//
				ELSE
					Mach_Control.DT_b.Error[5]:=TRUE;//叠负极片凸轮耦合时，隔膜平移轴即不在负极叠片位，也不在正极叠片位报警
					DP_Step0:=9992;	
				END_IF;							
			ELSIF Scan_TON[1].Q THEN
				Scan_TON[1].IN:=FALSE;	
				DP_Step0:=9993;
				DTPosError[4]:=TRUE;
			END_IF
		ELSE
			IF (Ca_Step0=0 OR Ca_Step0=6666) AND (Ca_Step3=0 OR Ca_Step3=6666) AND Scan_TON[2].Q THEN
				Scan_TON[2].IN:=FALSE;		
				DP_Step0:=9994;
				DTPosError[2]:=TRUE;
			END_IF
		END_IF
END_IF		

3010://负极搬运、叠片各轴在初始位，隔膜平移轴正极叠片位、正极叠片在放极片初始位
	IF NOT DP_SinStepe THEN
		Ca_CanIn5:=TRUE;
		IF Mach_Control.DT_b.SinStepMode THEN//单步调试模式
			DP_SinStepe:=TRUE;
		ELSE
			DP_SinStepe:=FALSE;	
		END_IF
		DP_Step0:=3020;	
	END_IF
3020:
	IF NOT DP_SinStepe THEN
		arrAxisCtrl[AxiseNo.VirAxisName.VirMain].Cmd	.bMoveAbs:=FALSE;	
		IF NOT Ca_CanIn5 THEN
			IF Mach_Control.DT_b.SinStepMode THEN//单步调试模式
				DP_SinStepe:=TRUE;
			ELSE
				DP_SinStepe:=FALSE;	
			END_IF
			DP_Step0:=3070;	
		ELSIF fbCaCamInCarryingLine2.bError OR  fbCaCamInDTCarryingLine.bError OR fbCaCamInDTCarryingUpDown.bError OR 
			fbCamInGMBuffer.bError OR fbCamInGMDanserMove.bError OR fbCamInVirGMDriver.bError OR fbAnCamInCarryingLine.bError OR 
			fbAnCamInDTCarryingLine.bError OR fbAnCamInCarryingWhirling.bError OR fbCamInLeftYDUpDown.bError OR fbCamInLeftYDLine.bError THEN
			Ca_CanIn5:=FALSE;
			Mach_Control.DT_b.Error[19]:=TRUE;//凸轮耦合报警
			DP_Step0:=9998;										
		END_IF
	END_IF
3030://负极搬运、叠片各轴在初始位，隔膜平移轴负极叠片位、正极叠片在取极片位
	IF NOT DP_SinStepe THEN
		Ca_CanIn6:=TRUE;
		IF Mach_Control.DT_b.SinStepMode THEN//单步调试模式
			DP_SinStepe:=TRUE;
		ELSE
			DP_SinStepe:=FALSE;	
		END_IF
		DP_Step0:=3040;
	END_IF
3040://判断凸轮耦合是否完成
	IF NOT DP_SinStepe THEN
		IF NOT Ca_CanIn6 THEN
			IF Mach_Control.DT_b.SinStepMode THEN//单步调试模式
				DP_SinStepe:=TRUE;
			ELSE
				DP_SinStepe:=FALSE;	
			END_IF
			DP_Step0:=3070;
		ELSIF  fbCaCamInCarryingLine2.bError OR fbCaCamInDTCarryingLine.bError OR 
			fbCaCamInDTCarryingUpDown.bError OR fbCamInLeftYDUpDown.bError OR 	fbCamInLeftYDLine.bError THEN										
			Ca_CanIn6:=FALSE;
			Mach_Control.DT_b.Error[19]:=TRUE;//凸轮耦合报警
			DP_Step0:=9995;		
		END_IF
	END_IF
3050://负极搬运、叠片各轴在初始位，隔膜平移轴正极叠片位、正极叠片在取极片位
	IF NOT DP_SinStepe THEN
		Ca_CanIn7:=TRUE;
		IF Mach_Control.DT_b.SinStepMode THEN//单步调试模式
			DP_SinStepe:=TRUE;
		ELSE
			DP_SinStepe:=FALSE;	
		END_IF
		DP_Step0:=3060;
	END_IF
3060:
	IF NOT DP_SinStepe THEN
			arrAxisCtrl[AxiseNo.VirAxisName.VirMain].Cmd	.bMoveAbs:=FALSE;	
			IF NOT Ca_CanIn7 THEN
				IF Mach_Control.DT_b.SinStepMode THEN//单步调试模式
					DP_SinStepe:=TRUE;
				ELSE
					DP_SinStepe:=FALSE;	
				END_IF																			
				DP_Step0:=3070;
			ELSIF fbCaCamInCarryingLine2.bError OR fbCaCamInDTCarryingLine.bError OR 
				fbCaCamInDTCarryingUpDown.bError OR fbCamInGMBuffer.bError OR fbCamInGMDanserMove.bError OR
				fbCamInVirGMDriver.bError OR fbCamInLeftYDUpDown.bError OR fbCamInLeftYDLine.bError  THEN
				Ca_CanIn7:=FALSE;
				Mach_Control.DT_b.Error[19]:=TRUE;//凸轮耦合报警
				DP_Step0:=9996;	
			END_IF
	END_IF

3070://判断负极叠片搬运机械手上是否有极片
	VirMain_TON.IN:=FALSE;
	DP_Step0:=3071;
	(*
	IF NOT DP_SinStepe THEN
		IF NOT arrCyCtrl[arrCyNo.ElectValveName.CaDTCarryingVacuum].Io.DIOnSwitch AND NOT Mach_Control.Ca_b.Ca_DPCarryingFalg  THEN	
			IF Mach_Control.DT_b.SinStepMode THEN//单步调试模式
				DP_SinStepe:=TRUE;
			ELSE
				DP_SinStepe:=FALSE;	
			END_IF
			DP_Step0:=3071;
		ELSE	
		  	Mach_Control.Ca_b.Error[28]:=TRUE; //负极叠片完空叠隔膜时，负极叠片搬运机械手真空检测有信号报警,请拿掉极片
		END_IF  
	END_IF	 
	*)
3071://主轴启动
	IF NOT DP_SinStepe THEN
		arrAxisCtrl[AxiseNo.VirAxisName.VirMain].Cmd	.bDynamitcsParSel:=2;
		arrAxisPar[AxiseNo.VirAxisName.VirMain].fTagatTime:=VirMain_TagatTime;
		arrAxisCtrl[AxiseNo.VirAxisName.VirMain].Cmd	.fPositon_of_Abs:=360;
		arrAxisCtrl[AxiseNo.VirAxisName.VirMain].Cmd	.bMoveAbs:=TRUE;	
		//fbCaCamInCarryingUpDown2OutCamFlge:=FALSE;//负极升降2凸轮解耦标记										
		IF  arrAxis[AxiseNo.VirAxisName.VirMain].Status.Moving OR arrAxisCtrl[AxiseNo.VirAxisName.VirMain].Status.fActPos>=10  THEN
			VirMain_TON.IN:=FALSE;
			arrAxisCtrl[AxiseNo.VirAxisName.VirMain].Cmd	.bMoveAbs:=FALSE;	
			DP_Step0:=3080;	
		ELSE
			IF NOT VirMain_TON.Q THEN
				VirMain_TON.IN:=TRUE;
			ELSE
				VirMain_TON.IN:=FALSE;
				Mach_Control.DT_b.Error[22]:=TRUE;//主轴启动超时报警
				DP_Step0:=10006;	
			END_IF	
		END_IF	
	END_IF	

END_CASE
END_IF


(**************************************************************************************电芯下料**************************************************************************************************************)
CASE DP_Step0 OF
2080:
IF arrAxis[AxiseNo.VirAxisName.VirMain].NcToPlc.SetPos>=234 AND arrAxis[AxiseNo.VirAxisName.VirMain].NcToPlc.SetPos<=240 THEN
	arrCyCtrl[arrCyNo.ElectValveName.AnDTCarryingVacuum].Cmd.bOFF:=FALSE;//正极叠片搬运升降真空关
     arrCyCtrl[arrCyNo.ElectValveName.AnDTCarryingVacuum].Cmd.bON:=TRUE;//正极叠片搬运升降真空关
	Mach_Control.An_b.An_DPCarryingFalg :=FALSE;//复位正极叠片搬运吸盘上有料标记																									
END_IF				
IF arrAxis[AxiseNo.VirAxisName.VirMain].NcToPlc.SetPos=360 AND  arrAxis[AxiseNo.VirAxisName.VirMain].Status.NotMoving  THEN
			Mach_Control.An_b.An_KDQuantited:=Mach_Control.An_b.An_KDQuantited +1;
			DP_Step1:=100;//解除耦合，主轴回零子程序
			arrAxisCtrl[AxiseNo.AxisName.DTUpDown].Cmd.fPosition_of_Rel:=-Par.stDT_date.SEPTA_Thickness;
			arrAxisPar[AxiseNo.AxisName.DTUpDown].fVelocity_of_Rel:=100;
			arrAxisCtrl[AxiseNo.AxisName.DTUpDown].Cmd.bMoveRel:=TRUE;
			DP_Step0:=0;
END_IF
	
(*2080:
	IF arrAxis[AxiseNo.VirAxisName.VirMain].NcToPlc.SetPos=360 AND  arrAxis[AxiseNo.VirAxisName.VirMain].Status.NotMoving  THEN
		Mach_Control.An_b.An_KDQuantited:=Mach_Control.An_b.An_KDQuantited +1;
		DPcount:=DPcount+1;	
		DP_Step1:=100;//解除耦合，主轴回零子程序
		arrAxisCtrl[AxiseNo.AxisName.DTUpDown].Cmd.fPosition_of_Rel:=-Par.stDT_date.SEPTA_Thickness;
		arrAxisPar[AxiseNo.AxisName.DTUpDown].fVelocity_of_Rel:=100;
		arrAxisCtrl[AxiseNo.AxisName.DTUpDown].Cmd.bMoveRel:=TRUE;
		DP_Step0:=0;
	END_IF*)


3080:

	IF arrAxis[AxiseNo.VirAxisName.VirMain].NcToPlc.SetPos=360 AND  arrAxis[AxiseNo.VirAxisName.VirMain].Status.NotMoving  THEN
		Mach_Control.Ca_b.Ca_KDQuantited:=Mach_Control.Ca_b.Ca_KDQuantited +1;
		DPcount:=DPcount+1;	
		DP_Step1:=100;//解除耦合，主轴回零子程序
		arrAxisCtrl[AxiseNo.AxisName.DTUpDown].Cmd.fPosition_of_Rel:=-Par.stDT_date.SEPTA_Thickness;
		arrAxisPar[AxiseNo.AxisName.DTUpDown].fVelocity_of_Rel:=100;
		arrAxisCtrl[AxiseNo.AxisName.DTUpDown].Cmd.bMoveRel:=TRUE;							
		DP_Step0:=0;
	END_IF		
END_CASE
END_ACTION

ACTION _01DT_Auto4:
IF Mach_Control.U.DT_iMode=1 THEN//在自动状态下
CASE DP_Step0 OF		
	6000://叠片完成，负极升降机械手回到安全位
			IF NOT DP_SinStepe THEN
						//负极取片2升降安全位
						IF arrAxisCtrl[AxiseNo.AxisName.CaCarryingUpDown2].Status.Homed AND arrAxisCtrl[AxiseNo.AxisName.CaCarryingUpDown2].Status.NoMoving AND 
							NOT arrAxisCtrl[AxiseNo.AxisName.CaCarryingUpDown2].Status.Error THEN
								IF arrAxisCtrl[AxiseNo.AxisName.CaCarryingUpDown2].Cmd.arrbRealPoint[4] THEN
										arrAxisCtrl[AxiseNo.AxisName.CaCarryingUpDown2].Cmd.iGoSetPos:=0;
								ELSE
									arrAxisCtrl[AxiseNo.AxisName.CaCarryingUpDown2].Cmd.iGoSetPos:=4;//负极搬运升降2移动至初始高度
								END_IF
						END_IF				
						//负极叠片取片升降等待位
						IF arrAxisCtrl[AxiseNo.AxisName.CaDTCarryingUpDown].Status.Homed AND arrAxisCtrl[AxiseNo.AxisName.CaDTCarryingUpDown].Status.NoMoving AND
							 NOT arrAxisCtrl[AxiseNo.AxisName.CaDTCarryingUpDown].Status.Error THEN
									IF arrAxisCtrl[AxiseNo.AxisName.CaDTCarryingUpDown].Cmd.arrbRealPoint[4] THEN
											arrAxisCtrl[AxiseNo.AxisName.CaDTCarryingUpDown].Cmd.iGoSetPos:=0;							
									ELSE
										arrAxisCtrl[AxiseNo.AxisName.CaDTCarryingUpDown].Cmd.iGoSetPos:=4;//负极叠片升降移动至等待高度
									END_IF
						END_IF
						
						IF 	arrAxisCtrl[AxiseNo.AxisName.CaCarryingUpDown2].Cmd.arrbRealPoint[4]  AND  arrAxisCtrl[AxiseNo.AxisName.CaCarryingUpDown2].Status.NoMoving AND 
								arrAxisCtrl[AxiseNo.AxisName.CaDTCarryingUpDown].Cmd.arrbRealPoint[4] 	AND arrAxisCtrl[AxiseNo.AxisName.CaDTCarryingUpDown].Status.NoMoving THEN
								IF Mach_Control.DT_b.SinStepMode THEN//单步调试模式
											DP_SinStepe:=TRUE;
								ELSE
											DP_SinStepe:=FALSE;	
								END_IF
								DP_Step0:=6010;
					END_IF
			END_IF
		6010://判断主轴是否停止、是否在初始位、是否有轴在耦合中
			IF NOT DP_SinStepe THEN
				IF CA_CarryingPos2 THEN
					IF arrAxisCtrl[AxiseNo.VirAxisName.VirMain].Status.NoMoving AND arrAxis[AxiseNo.VirAxisName.VirMain].NcToPlc.ActPos=0 AND NOT DT_AxiseCoupling THEN
						DT_SingeMode();//单步选择						
						DP_Step0:=6012;
					ELSE
						DP_Step1:=100;//调用主轴回初始位子程序
						DT_SingeMode();//单步选择							
						DP_Step0:=6011;
					END_IF
				ELSIF  CA_CarryingPos1 THEN
					DP_Step0:=6014;
				END_IF	
			END_IF
					
		6011://判断主轴的模长的当前位置是否为0
			IF NOT DP_SinStepe THEN
				IF DP_Step1=6666 AND arrAxisCtrl[AxiseNo.VirAxisName.VirMain].Status.NoMoving AND arrAxis[AxiseNo.VirAxisName.VirMain].NcToPlc.ActPos=0 AND NOT DT_AxiseCoupling THEN
					DT_SingeMode();//单步选择						
					DP_Step0:=6012;
				END_IF
			END_IF		

		6012:
			//负极送片搬运平移
				fbCaCamInCarryingLine2.ParCamIn.SlaveScaling:=-1;
				fbCaCamInCarryingLine2.bCamInExecute:=TRUE;								
		        fbCaCamInCarryingUpDown2.iTableSel:=3;    //20240528SJ
	            fbCaCamInCarryingUpDown2.bCamInExecute:=TRUE;		
				
			//负极叠台搬运平移
				fbCaCamInDTCarryingLine.ParCamIn.SlaveScaling:=-1;
				fbCaCamInDTCarryingLine.bCamInExecute:=TRUE;	
			    fbCaCamInDTCarryingUpDown.iTableSel:=3;   //20240528SJ
	            fbCaCamInDTCarryingUpDown.bCamInExecute:=TRUE;
				
			//负极叠片升降轴放片凸轮耦合
				//fbCaCamInDTCarryingUpDown.iTableSel:=2;
				//fbCaCamInDTCarryingUpDown.bCamInExecute:=TRUE;		
														  
			IF fbCaCamInCarryingLine2.bInSync AND fbCaCamInDTCarryingLine.bInSync AND  fbCaCamInCarryingUpDown2.bInSync AND fbCaCamInDTCarryingUpDown.bInSync   THEN   
				DT_SingeMode();//单步选择		
				DP_Step0:=6013;
			ELSIF fbCaCamInCarryingLine2.bError  OR  fbCaCamInDTCarryingLine.bError  OR 
                    fbCaCamInCarryingUpDown2.bError OR fbCaCamInDTCarryingUpDown.bError   THEN   
				Mach_Control.DT_b.Error[19]:=TRUE;//凸轮耦合报警
			END_IF	
		6074:	
			IF arrAxis[AxiseNo.VirAxisName.VirMain].NcToPlc.SetPos=360 AND  arrAxis[AxiseNo.VirAxisName.VirMain].Status.NotMoving THEN 
				DP_Step1:=100;
				DP_Step0:=6075;	
			END_IF
		  
		6075:  
			IF DP_Step1=6666 THEN	
				DP_Step0:=6014;						
			END_IF		
		  
		6014:
			IF arrAxisCtrl[AxiseNo.VirAxisName.VirMain].Status.NoMoving AND arrAxis[AxiseNo.VirAxisName.VirMain].NcToPlc.ActPos=0 AND NOT DT_AxiseCoupling 
				AND CA_CarryingPos1 THEN
				DP_Step0:=6015;	
			ELSIF  DT_AxiseCoupling THEN
				DP_Step1:=100;
				DP_Step0:=6075;	
			END_IF  
	(*
				IF NOT DP_SinStepe THEN
					//负极取片2平移取片位
											IF arrAxisCtrl[AxiseNo.AxisName.CaCarryingUpDown2].Cmd.arrbRealPoint[5] AND arrAxisCtrl[AxiseNo.AxisName.CaCarryingLine2].Status.Homed AND
												 arrAxisCtrl[AxiseNo.AxisName.CaCarryingLine2].Status.NoMoving AND NOT arrAxisCtrl[AxiseNo.AxisName.CaCarryingLine2].Status.Error THEN
													IF arrAxisCtrl[AxiseNo.AxisName.CaCarryingLine2].Cmd.arrbRealPoint[1] THEN
															arrAxisCtrl[AxiseNo.AxisName.CaCarryingLine2].Cmd.iGoSetPos:=0;					
													ELSE
														arrAxisCtrl[AxiseNo.AxisName.CaCarryingLine2].Cmd.iGoSetPos:=1;//负极搬运平移2移动至初始位取流水线上的极片
													END_IF
											END_IF
					//负极叠片平移取片位
										IF TailCurlSEPTA_SafePos  AND arrAxisCtrl[AxiseNo.AxisName.CaDTCarryingUpDown].Cmd.arrbRealPoint[4] AND arrAxisCtrl[AxiseNo.AxisName.CaDTCarryingLine].Status.Homed AND
											 arrAxisCtrl[AxiseNo.AxisName.CaDTCarryingLine].Status.NoMoving AND NOT arrAxisCtrl[AxiseNo.AxisName.CaDTCarryingLine].Status.Error THEN
												IF arrAxisCtrl[AxiseNo.AxisName.CaDTCarryingLine].Cmd.arrbRealPoint[1] THEN
														arrAxisCtrl[AxiseNo.AxisName.CaDTCarryingLine].Cmd.iGoSetPos:=0;
												ELSE
													arrAxisCtrl[AxiseNo.AxisName.CaDTCarryingLine].Cmd.iGoSetPos:=1;//负极叠片平移至初始位
												END_IF
										END_IF
										
										IF 	arrAxisCtrl[AxiseNo.AxisName.CaCarryingLine2].Cmd.arrbRealPoint[1] AND 	arrAxisCtrl[AxiseNo.AxisName.CaCarryingLine2].Status.NoMoving AND 
													arrAxisCtrl[AxiseNo.AxisName.CaDTCarryingLine].Cmd.arrbRealPoint[1] AND 	arrAxisCtrl[AxiseNo.AxisName.CaDTCarryingLine].Status.NoMoving THEN
													IF Mach_Control.DT_b.SinStepMode THEN//单步调试模式
																DP_SinStepe:=TRUE;
													ELSE
																DP_SinStepe:=FALSE;	
													END_IF
													DP_Step0:=6015;	
										//ELSIF  THEN											
										END_IF
				END_IF
	*)			
		6015:
			IF NOT DP_SinStepe THEN
					//负极叠片升降避让位
					IF arrAxisCtrl[AxiseNo.AxisName.CaDTCarryingUpDown].Status.Homed AND arrAxisCtrl[AxiseNo.AxisName.CaDTCarryingUpDown].Status.NoMoving AND
						 NOT arrAxisCtrl[AxiseNo.AxisName.CaDTCarryingUpDown].Status.Error THEN
						IF arrAxisCtrl[AxiseNo.AxisName.CaDTCarryingUpDown].Cmd.arrbRealPoint[5] THEN
								arrAxisCtrl[AxiseNo.AxisName.CaDTCarryingUpDown].Cmd.iGoSetPos:=0;							
						ELSE
							arrAxisCtrl[AxiseNo.AxisName.CaDTCarryingUpDown].Cmd.iGoSetPos:=5;//负极叠片升降移动至避让高度
						END_IF
					END_IF
					
					IF 	arrAxisCtrl[AxiseNo.AxisName.CaDTCarryingUpDown].Cmd.arrbRealPoint[5] 	AND arrAxisCtrl[AxiseNo.AxisName.CaDTCarryingUpDown].Status.NoMoving THEN
						IF Mach_Control.DT_b.SinStepMode THEN//单步调试模式
							DP_SinStepe:=TRUE;
						ELSE
							DP_SinStepe:=FALSE;	
						END_IF
						DP_Step0:=6016;
				END_IF
			END_IF
END_CASE
END_IF


CASE DP_Step0 OF
	6013:
		IF NOT DP_SinStepe THEN
			 arrAxisCtrl[AxiseNo.VirAxisName.VirMain].Cmd.bDynamitcsParSel:=2;	
			 arrAxisPar[AxiseNo.VirAxisName.VirMain].fTagatTime:=VirMain_TagatTime;
			 arrAxisCtrl[AxiseNo.VirAxisName.VirMain].Cmd.fPositon_of_Abs:=360;
			 arrAxisCtrl[AxiseNo.VirAxisName.VirMain].Cmd.bMoveAbs:=TRUE;			
			IF  arrAxis[AxiseNo.VirAxisName.VirMain].Status.Moving OR arrAxisCtrl[AxiseNo.VirAxisName.VirMain].Status.fActPos>=5  THEN		
				arrAxisCtrl[AxiseNo.VirAxisName.VirMain].Cmd.bMoveAbs:=FALSE;
				Ca_TON[2].IN:=FALSE;                               	
				DP_Step0:=6074;	
				//Ca_StandbyStep1:=300;  //取消调用负极送片搬运取流水线极片
				//Ca_StandbyStep5:=400;
			ELSE
				IF NOT Ca_TON[2].Q THEN
					Ca_TON[2].IN:=TRUE;
				ELSE
				Ca_TON[2].IN:=FALSE;
					Mach_Control.DT_b.Error[22]:=TRUE;//主轴启动超时报警
					arrAxisCtrl[AxiseNo.VirAxisName.VirMain].Cmd	.bMoveAbs:=FALSE;	
				END_IF
			END_IF	
		END_IF	
					
	6016://纠偏平台回原
		 IF arrAxisCtrl[AxiseNo.AxisName.AnDTCarryingUpDown].Cmd.arrbRealPoint[4] AND arrAxisCtrl[AxiseNo.AxisName.CaDTCarryingUpDown].Cmd.arrbRealPoint[5]  THEN
			 DP_Step11:=100;//正极纠偏平台回原
			 DP_Step12:=100;//负极纠偏平台回原
			 DP_Step0:=6020;
		 END_IF


	6020:
				IF Mach_Control.DT_b.DT_Oerhang_Z<>2 OR   Mach_Control.DT_b.DT_Overhang THEN
					CellMemory[Mach_Control.DT_b.DT_Memory].Hough:=1;
					DP_Step0:=6025;
					NN:=0;
				ELSE 
					CellMemory[Mach_Control.DT_b.DT_Memory].Hough:=2;
					DP_Step0:=6024;
				END_IF
				
	6024:
				NN:=NN+1;
				DP_Step0:=6025;			
																
	6025:
			Mach_Control.DT_b.DT_amount:=Mach_Control.DT_b.DT_amount+1;
			CellMemory[Mach_Control.DT_b.DT_Memory].Cell:=TRUE;	
			CellMemory[Mach_Control.DT_b.DT_Memory].DT_station_No:=Mach_Control.DT_b.DT_No;
			CellMemory[Mach_Control.DT_b.DT_Memory].DT_speed:=Par.stDT_date.SinglePosTime;
			CellMemory[Mach_Control.DT_b.DT_Memory].An_Quantity:=Mach_Control.An_b.An_Quantited;
			CellMemory[Mach_Control.DT_b.DT_Memory].Ca_Quantity:=Mach_Control.Ca_b.Ca_Quantited;
			//CellMemory[Mach_Control.DT_b.DT_Memory].DiaphragmUnwindingTension:=LIMIT(150,Mach_Control.DT_b.DiaphragmUnwindingTension,250);	
            // CellMemory[Mach_Control.DT_b.DT_Memory].DiaphragmUnwindingTension:=CellMemory[Mach_Control.DT_b.DT_Memory].Chipdata[210].GMlapTen;				
			//CellMemory[Mach_Control.DT_b.DT_Memory].DiaphragmUnwindingTension_max:=ABS(Mach_Control.DT_b.DiaphragmUnwindingTension+10);	
			//CellMemory[Mach_Control.DT_b.DT_Memory].DiaphragmUnwindingTension_min:=ABS(Mach_Control.DT_b.DiaphragmUnwindingTension-4);	
			//CellMemory[Mach_Control.DT_b.DT_Memory].DiaphragmUnwindingTension_ave:=ABS(Mach_Control.DT_b.DiaphragmUnwindingTension+5);	
			//[Mach_Control.DT_b.DT_Memory].DiaphragmUnwindingTension_set:=ABS(Mach_Control.DT_b.DiaphragmUnwindingTension);
	
            CellMemory[Mach_Control.DT_b.DT_Memory].DiaphragmUnwindingTension:=LIMIT(150,CellMemory[Mach_Control.DT_b.DT_Memory].Chipdata[210].GMlapTen,250);				
			CellMemory[Mach_Control.DT_b.DT_Memory].DiaphragmUnwindingTension_max:=LIMIT(150,CellMemory[Mach_Control.DT_b.DT_Memory].Chipdata[210].GMlapTen+10,250);	
			CellMemory[Mach_Control.DT_b.DT_Memory].DiaphragmUnwindingTension_min:=LIMIT(150,CellMemory[Mach_Control.DT_b.DT_Memory].Chipdata[210].GMlapTen-4,250);	
			CellMemory[Mach_Control.DT_b.DT_Memory].DiaphragmUnwindingTension_ave:=LIMIT(150,CellMemory[Mach_Control.DT_b.DT_Memory].Chipdata[210].GMlapTen+5,250);	
			CellMemory[Mach_Control.DT_b.DT_Memory].DiaphragmUnwindingTension_set:=LIMIT(150,CellMemory[Mach_Control.DT_b.DT_Memory].Chipdata[210].GMlapTen,250);	
			
			CellMemory[Mach_Control.DT_b.DT_Memory].Put_Time :=Mach_Control.DT_b.Put_time;
			CellMemory[Mach_Control.DT_b.DT_Memory].Machine_No:=Mach_Control.DT_b.Machine_No;
			CellMemory[Mach_Control.DT_b.DT_Memory].Cell_CCD_No:=CCD.Over.Finish.stCellNo;
			CellMemory[Mach_Control.DT_b.DT_Memory].BlueGlue:=1;
			
			CellMemory[Mach_Control.DT_b.DT_Memory].An_stuff_No:=Par.stDT_date.An_stuff_No;
			CellMemory[Mach_Control.DT_b.DT_Memory].Ca_stuff_No:=Par.stDT_date.Ca_stuff_No;
			CellMemory[Mach_Control.DT_b.DT_Memory].Diaphragm_No:=Par.stDT_date.Diaphragm_No;
			CellMemory[Mach_Control.DT_b.DT_Memory].PostiveCode:=CellMemory[Mach_Control.DT_b.DT_Memory].An_MQ_Slice[Mach_Control.An_b.An_Quantited].Code;//正极片条码
			CellMemory[Mach_Control.DT_b.DT_Memory].NegativeCode:=CellMemory[Mach_Control.DT_b.DT_Memory].Ca_MQ_Slice[Mach_Control.Ca_b.Ca_Quantited].Code;//负极片条码
		
		    CellMemory[Mach_Control.DT_b.DT_Memory].LYDLineinitPos:=arrAxisPar[AxiseNo.AxisName.LeftYDLine].arrTargetPoint[1];
			CellMemory[Mach_Control.DT_b.DT_Memory].LYDLineOpenPos :=arrAxisPar[AxiseNo.AxisName.LeftYDLine].arrTargetPoint[2];
			CellMemory[Mach_Control.DT_b.DT_Memory].LYDLinepressL :=arrAxisPar[AxiseNo.AxisName.LeftYDLine].arrTargetPoint[12];
			CellMemory[Mach_Control.DT_b.DT_Memory].RYDLineinitPos:=arrAxisPar[AxiseNo.AxisName.RightYDLine].arrTargetPoint[1];
			CellMemory[Mach_Control.DT_b.DT_Memory].RYDLineOpenPos :=arrAxisPar[AxiseNo.AxisName.RightYDLine].arrTargetPoint[2];
			CellMemory[Mach_Control.DT_b.DT_Memory].RYDLinepressL :=arrAxisPar[AxiseNo.AxisName.RightYDLine].arrTargetPoint[12];
			CellMemory[Mach_Control.DT_b.DT_Memory].LYDUpDowninitPos:=arrAxisPar[AxiseNo.AxisName.LeftYDUpDown].arrTargetPoint[1];
			CellMemory[Mach_Control.DT_b.DT_Memory].LYDUpDownOpenPos :=arrAxisPar[AxiseNo.AxisName.LeftYDUpDown].arrTargetPoint[2];
			CellMemory[Mach_Control.DT_b.DT_Memory].LYDUpDownOpenH:=arrAxisPar[AxiseNo.AxisName.LeftYDUpDown].arrTargetPoint[11];
			CellMemory[Mach_Control.DT_b.DT_Memory].LYDUpDownKnifeH:=arrAxisPar[AxiseNo.AxisName.LeftYDUpDown].arrTargetPoint[12];
			CellMemory[Mach_Control.DT_b.DT_Memory].RYDUpDowninitPos :=arrAxisPar[AxiseNo.AxisName.RightYDUpDown].arrTargetPoint[1];
			CellMemory[Mach_Control.DT_b.DT_Memory].RYDUpDownOpenPos :=arrAxisPar[AxiseNo.AxisName.RightYDUpDown].arrTargetPoint[2];
			CellMemory[Mach_Control.DT_b.DT_Memory].RYDUpDownOpenH:=arrAxisPar[AxiseNo.AxisName.RightYDUpDown].arrTargetPoint[11];
			CellMemory[Mach_Control.DT_b.DT_Memory].RYDUpDownKnifeH:=arrAxisPar[AxiseNo.AxisName.RightYDUpDown].arrTargetPoint[12];
			CellMemory[Mach_Control.DT_b.DT_Memory].DTandescendh:=Par.stDT_date.An_Thickness+Par.stDT_date.SEPTA_Thickness+Par.stDT_date.Pole_ThicknessCom;
			CellMemory[Mach_Control.DT_b.DT_Memory].DTcadescendh:=Par.stDT_date.Ca_Thickness+Par.stDT_date.SEPTA_Thickness+Par.stDT_date.Pole_ThicknessCom;
		
			
			IF Mach_Control.DT_b.DT_DebugMode THEN
			   CellMemory[Mach_Control.DT_b.DT_Memory].DTDebugMode:=TRUE;
			END_IF
			
			IF Mach_Control.DT_b.Overhang_TF THEN
			CellMemory[Mach_Control.DT_b.DT_Memory].Overhang_TF:=TRUE;
			ELSE
			CellMemory[Mach_Control.DT_b.DT_Memory].Overhang_TF:=FALSE;	
			END_IF
			DP_Step0:=6030;	

					
	6030:			
				Mach_Control.DT_b.Overhang_TF:=FALSE;	
				Mach_Control.DT_b.OffloadRequest:=TRUE;//叠电芯完成，请求下电芯
				DP_Step0:=6040;	
	6040://
		IF Mach_Control.DT_b.OffloadDone THEN
			bFirstFoldFinish[1]:=FALSE;//首层隔膜空叠
			bFirstFoldFinish[2]:=FALSE;//正常电芯空叠隔膜
			bFirstFoldFinish[3]:=FALSE;//接带、黄标空叠隔膜
			bEmptyFoldMark[1]:=FALSE;//进入空叠流程
			bEmptyFoldMark[2]:=FALSE;//进入空叠流程
			bEmptyFoldMark[3]:=FALSE;//进入空叠流程	
			Mach_Control.An_b.An_FirstFoldCnt:=0;
			Mach_Control.Ca_b.Ca_FirstFoldCnt:=0;
			Mach_Control.DT_b.OffloadRequest:=FALSE;//叠电芯完成，请求下电芯
			Mach_Control.An_b.An_Quantited:=0;
			Mach_Control.Ca_b.Ca_Quantited:=0;
			Mach_Control.An_b.An_KDQuantited :=0;
			Mach_Control.Ca_b.Ca_KDQuantited:=0;
			Mach_Control.DT_b.OffloadDone:=FALSE;
			OversequelNG:=FALSE;	
			DP_Step0:=6041;	
		END_IF

	6041://负极叠台升降、取片升降到等待高度等待耦合
		IF arrAxisCtrl[AxiseNo.AxisName.CaDTCarryingUpDown].Cmd.arrbRealPoint[4] THEN
			arrAxisCtrl[AxiseNo.AxisName.CaDTCarryingUpDown].Cmd.iGoSetPos:=0;				
		ELSE
			arrAxisCtrl[AxiseNo.AxisName.CaDTCarryingUpDown].Cmd.iGoSetPos:=4;//负极叠片升降移动至取片位
		END_IF
		IF arrAxisCtrl[AxiseNo.AxisName.CaCarryingUpDown2].Cmd.arrbRealPoint[4] THEN
			arrAxisCtrl[AxiseNo.AxisName.CaCarryingUpDown2].Cmd.iGoSetPos:=0;				
		ELSE
			arrAxisCtrl[AxiseNo.AxisName.CaCarryingUpDown2].Cmd.iGoSetPos:=4;//负极叠片升降移动至取片位
		END_IF
		IF  arrAxisCtrl[AxiseNo.AxisName.CaDTCarryingUpDown].Cmd.arrbRealPoint[4] AND arrAxisCtrl[AxiseNo.AxisName.CaCarryingUpDown2].Cmd.arrbRealPoint[4] THEN
			DP_Step0:=6042;
		END_IF
	
	6042://	等待纠偏平台回原完成		
			IF DP_Step11=6666 AND DP_Step12=6666 THEN
			   DP_Step0:=0;
			END_IF															
END_CASE
END_ACTION

ACTION _01DT_Auto5:

//
IF Ca_CanIn1 THEN  //OK
//负到正_负极搬运平移2轴凸轮耦合
	fbCaCamInCarryingLine2.ParCamIn.SlaveScaling:=1;
	fbCaCamInCarryingLine2.bCamInExecute:=TRUE;
//负到正_负极搬运升降2轴放片凸轮耦合
	fbCaCamInCarryingUpDown2.iTableSel:=2;
	fbCaCamInCarryingUpDown2.bCamInExecute:=TRUE;
//负到正_负极叠片平移轴凸轮耦合
	fbCaCamInDTCarryingLine.ParCamIn.SlaveScaling:=1;
	fbCaCamInDTCarryingLine.bCamInExecute:=TRUE;
//负到正_负极叠片升降轴放片凸轮耦合
	fbCaCamInDTCarryingUpDown.iTableSel:=2;
	fbCaCamInDTCarryingUpDown.bCamInExecute:=TRUE;
//叠台左压刀升降凸轮耦合
	//fbCamInLeftYDUpDown.bCamInExecute:=TRUE;
//叠台左压刀开合凸轮耦合
	//fbCamInLeftYDLine.bCamInExecute:=TRUE;
IF arrAxisCtrl[AxiseNo.AxisName.LeftYDLine].Cmd.arrbRealPoint[1] THEN
	fbCamInLeftYDUpDown.iTableSel:=1;
	fbCamInLeftYDLine.iTableSel:=1;
	fbCamInLeftYDUpDown.bCamInExecute:=TRUE;
	fbCamInLeftYDLine.bCamInExecute:=TRUE;	
ELSIF arrAxisCtrl[AxiseNo.AxisName.LeftYDLine].Cmd.arrbRealPoint[2] THEN	
	fbCamInLeftYDUpDown.iTableSel:=2;
	fbCamInLeftYDLine.iTableSel:=2;
	fbCamInLeftYDUpDown.bCamInExecute:=TRUE;
	fbCamInLeftYDLine.bCamInExecute:=TRUE;		
END_IF
//判断凸轮耦合是否完成
	IF 	fbCaCamInCarryingLine2.bInSync AND fbCaCamInCarryingUpDown2	.bInSync AND 	fbCaCamInDTCarryingLine.bInSync AND 	fbCaCamInDTCarryingUpDown.bInSync AND 
		fbCamInLeftYDUpDown.bInSync AND fbCamInLeftYDLine.bInSync 	 THEN
		Ca_CanIn1:=FALSE;
		//DP_Step0:=141;
	END_IF	
END_IF
//
IF Ca_CanIn2 THEN //OK
//负到正_负极搬运平移2轴凸轮耦合
	fbCaCamInCarryingLine2.ParCamIn.SlaveScaling:=1;
	fbCaCamInCarryingLine2.bCamInExecute:=TRUE;						
//负到正_负极搬运升降2轴放片凸轮耦合
	fbCaCamInCarryingUpDown2.iTableSel:=2;
	fbCaCamInCarryingUpDown2.bCamInExecute:=TRUE;
//负到正_负极叠片平移轴凸轮耦合
	fbCaCamInDTCarryingLine.ParCamIn.SlaveScaling:=1;
	fbCaCamInDTCarryingLine.bCamInExecute:=TRUE;						
//负到正_负极叠片升降轴放片凸轮耦合
	fbCaCamInDTCarryingUpDown.iTableSel:=2;
	fbCaCamInDTCarryingUpDown.bCamInExecute:=TRUE;
//负到正_缓存轴凸轮耦合	
	fbCamInGMBuffer.iTableSel:=2;
	fbCamInGMBuffer.bCamInExecute:=TRUE;
//负到正_隔膜平移轴凸轮耦合
	fbCamInGMDanserMove.iTableSel:=2;
	fbCamInGMDanserMove.bCamInExecute:=TRUE;

//负到正_放卷虚轴凸轮耦合
	fbCamInVirGMDriver.iTableSel:=2;
	fbCamInVirGMDriver.bCamInExecute:=TRUE;
//叠台左压刀升降凸轮耦合
	//fbCamInLeftYDUpDown.bCamInExecute:=TRUE;
//叠台左压刀开合凸轮耦合
	//fbCamInLeftYDLine.bCamInExecute:=TRUE;	
IF arrAxisCtrl[AxiseNo.AxisName.LeftYDLine].Cmd.arrbRealPoint[1] THEN
	fbCamInLeftYDUpDown.iTableSel:=1;
	fbCamInLeftYDLine.iTableSel:=1;
	fbCamInLeftYDUpDown.bCamInExecute:=TRUE;
	fbCamInLeftYDLine.bCamInExecute:=TRUE;	
ELSIF arrAxisCtrl[AxiseNo.AxisName.LeftYDLine].Cmd.arrbRealPoint[2] THEN	
	fbCamInLeftYDUpDown.iTableSel:=2;
	fbCamInLeftYDLine.iTableSel:=2;
	fbCamInLeftYDUpDown.bCamInExecute:=TRUE;
	fbCamInLeftYDLine.bCamInExecute:=TRUE;		
END_IF
					
//判断凸轮耦合是否完成
	IF fbCaCamInCarryingLine2.bInSync AND fbCaCamInCarryingUpDown2.bInSync AND fbCaCamInDTCarryingLine.bInSync AND
		fbCaCamInDTCarryingUpDown.bInSync AND fbCamInGMBuffer.bInSync AND fbCamInGMDanserMove.bInSync AND 
		fbCamInVirGMDriver.bInSync AND fbCamInLeftYDUpDown.bInSync AND fbCamInLeftYDLine.bInSync    THEN								
		Ca_CanIn2:=FALSE;
		//DP_Step0:=141;
	END_IF
END_IF
//
IF Ca_CanIn3 THEN    //OK
//负到正_负极搬运平移2轴凸轮耦合
	fbCaCamInCarryingLine2.ParCamIn.SlaveScaling:=1;
	fbCaCamInCarryingLine2.bCamInExecute:=TRUE;									
//负到正_负极搬运升降2轴放片凸轮耦合
	fbCaCamInCarryingUpDown2.iTableSel:=2;
	fbCaCamInCarryingUpDown2.bCamInExecute:=TRUE;
//负到正_负极叠片平移轴凸轮耦合
	fbCaCamInDTCarryingLine.ParCamIn.SlaveScaling:=1;
	fbCaCamInDTCarryingLine.bCamInExecute:=TRUE;							
//负到正_负极叠片升降轴放片凸轮耦合
	fbCaCamInDTCarryingUpDown.iTableSel:=2;
	fbCaCamInDTCarryingUpDown.bCamInExecute:=TRUE;						
//负到正_正极搬运平移轴凸轮耦合
	fbAnCamInCarryingLine.ParCamIn.SlaveScaling:=-1;
	fbAnCamInCarryingLine.bCamInExecute:=TRUE;
//负到正_正极搬运升降轴取片凸轮耦合	
	fbAnCamInCarryingUpDown.iTableSel:=1;	
	fbAnCamInCarryingUpDown.bCamInExecute:=TRUE;
//负到正_正极叠片平移轴凸轮耦合
	fbAnCamInDTCarryingLine.ParCamIn.SlaveScaling:=-1;
	fbAnCamInDTCarryingLine.bCamInExecute:=TRUE;
//负到正_正极叠片升降轴取片凸轮耦合
	fbAnCamInDTCarryingUpDown.iTableSel:=1;
	fbAnCamInDTCarryingUpDown.bCamInExecute:=TRUE;
//负到正_正极搬运旋转轴凸轮耦合	
	fbAnCamInCarryingWhirling.ParCamIn.SlaveScaling:=-1;
	fbAnCamInCarryingWhirling.bCamInExecute:=TRUE;
//叠台左压刀升降凸轮耦合
	//fbCamInLeftYDUpDown.bCamInExecute:=TRUE;
//叠台左压刀开合凸轮耦合
	//fbCamInLeftYDLine.bCamInExecute:=TRUE;
IF arrAxisCtrl[AxiseNo.AxisName.LeftYDLine].Cmd.arrbRealPoint[1] THEN
	fbCamInLeftYDUpDown.iTableSel:=1;
	fbCamInLeftYDLine.iTableSel:=1;
	fbCamInLeftYDUpDown.bCamInExecute:=TRUE;
	fbCamInLeftYDLine.bCamInExecute:=TRUE;	
ELSIF arrAxisCtrl[AxiseNo.AxisName.LeftYDLine].Cmd.arrbRealPoint[2] THEN	
	fbCamInLeftYDUpDown.iTableSel:=2;
	fbCamInLeftYDLine.iTableSel:=2;
	fbCamInLeftYDUpDown.bCamInExecute:=TRUE;
	fbCamInLeftYDLine.bCamInExecute:=TRUE;		
END_IF									
//	判断凸轮耦合是否完成
	IF fbCaCamInCarryingLine2.bInSync AND fbCaCamInCarryingUpDown2.bInSync AND fbCaCamInDTCarryingLine.bInSync AND fbCaCamInDTCarryingUpDown.bInSync AND 
		fbAnCamInCarryingLine.bInSync AND fbAnCamInCarryingUpDown.bInSync AND fbAnCamInDTCarryingLine.bInSync AND fbAnCamInDTCarryingUpDown.bInSync AND
		fbAnCamInCarryingWhirling.bInSync AND fbCamInLeftYDUpDown.bInSync AND fbCamInLeftYDLine.bInSync THEN
		Ca_CanIn3:=FALSE;
		//DP_Step0:=161;
	END_IF				
END_IF

//
IF Ca_CanIn4 THEN    //OK
//负到正_负极搬运平移2轴凸轮耦合
	fbCaCamInCarryingLine2.ParCamIn.SlaveScaling:=1;
	fbCaCamInCarryingLine2.bCamInExecute:=TRUE;							
//负到正_负极搬运升降2轴放片凸轮耦合
	fbCaCamInCarryingUpDown2.iTableSel:=2;
	fbCaCamInCarryingUpDown2.bCamInExecute:=TRUE;					
//负到正_负极叠片平移轴凸轮耦合
	fbCaCamInDTCarryingLine.ParCamIn.SlaveScaling:=1;
	fbCaCamInDTCarryingLine.bCamInExecute:=TRUE;							
//负到正_负极叠片升降轴放片凸轮耦合
	fbCaCamInDTCarryingUpDown.iTableSel:=2;
	fbCaCamInDTCarryingUpDown.bCamInExecute:=TRUE;		
//负到正_缓存轴凸轮耦合
	fbCamInGMBuffer.iTableSel:=2;
	fbCamInGMBuffer.bCamInExecute:=TRUE;					
//负到正_隔膜平移轴凸轮耦合
	fbCamInGMDanserMove.iTableSel:=2;
	fbCamInGMDanserMove.bCamInExecute:=TRUE;

	
//负到正_放卷虚轴凸轮耦合		
	fbCamInVirGMDriver.iTableSel:=2;
	fbCamInVirGMDriver.bCamInExecute:=TRUE;		
//负到正_正极搬运平移轴凸轮耦合	
	fbAnCamInCarryingLine.ParCamIn.SlaveScaling:=-1;
	fbAnCamInCarryingLine.bCamInExecute:=TRUE;															
//负到正_正极搬运升降轴取片凸轮耦合
	IF NOT DP_CheseCam THEN//???????????????
		fbAnCamInCarryingUpDown.iTableSel:=3;  //20240528SJ
		fbAnCamInCarryingUpDown.bCamInExecute:=TRUE;
	ELSE
		fbAnCamInCarryingUpDown.iTableSel:=3;  //20240528SJ
		fbAnCamInCarryingUpDown.bCamInExecute:=TRUE;		
	END_IF
	
//负到正_正极叠片平移轴凸轮耦合
	fbAnCamInDTCarryingLine.ParCamIn.SlaveScaling:=-1;
	fbAnCamInDTCarryingLine.bCamInExecute:=TRUE;	
//负到正_正极叠片升降轴取片凸轮耦合
IF NOT DP_CheseCam AND iAnCamInSel2=1 THEN
	fbAnCamInDTCarryingUpDown.iTableSel:=1;
	fbAnCamInDTCarryingUpDown.bCamInExecute:=TRUE;
ELSE
	fbAnCamInDTCarryingUpDown.iTableSel:=3;//20240528SJ
	fbAnCamInDTCarryingUpDown.bCamInExecute:=TRUE;	
END_IF

//负到正_正极搬运旋转轴凸轮耦合
	fbAnCamInCarryingWhirling.ParCamIn.SlaveScaling:=-1;
	fbAnCamInCarryingWhirling.bCamInExecute:=TRUE;
//叠台左压刀升降凸轮耦合
	//fbCamInLeftYDUpDown.bCamInExecute:=TRUE;
//叠台左压刀开合凸轮耦合
	//fbCamInLeftYDLine.bCamInExecute:=TRUE;	
IF arrAxisCtrl[AxiseNo.AxisName.LeftYDLine].Cmd.arrbRealPoint[1] THEN
	fbCamInLeftYDUpDown.iTableSel:=1;
	fbCamInLeftYDLine.iTableSel:=1;
	fbCamInLeftYDUpDown.bCamInExecute:=TRUE;
	fbCamInLeftYDLine.bCamInExecute:=TRUE;	
ELSIF arrAxisCtrl[AxiseNo.AxisName.LeftYDLine].Cmd.arrbRealPoint[2] THEN	
	fbCamInLeftYDUpDown.iTableSel:=2;
	fbCamInLeftYDLine.iTableSel:=2;
	fbCamInLeftYDUpDown.bCamInExecute:=TRUE;
	fbCamInLeftYDLine.bCamInExecute:=TRUE;		
END_IF				
//判断凸轮是否耦合完成
	IF fbCaCamInCarryingLine2.bInSync AND fbCaCamInCarryingUpDown2.bInSync AND fbCaCamInDTCarryingLine.bInSync AND  fbCaCamInDTCarryingUpDown.bInSync AND
	   fbCamInGMBuffer.bInSync AND fbCamInGMDanserMove.bInSync AND  fbCamInVirGMDriver.bInSync AND
		 fbAnCamInCarryingLine.bInSync AND fbAnCamInCarryingUpDown.bInSync AND  fbAnCamInCarryingWhirling.bInSync AND
		 fbAnCamInDTCarryingLine.bInSync AND ((fbAnCamInDTCarryingUpDown.bInSync AND  iAnCamInSel2=1 ) OR  (iAnCamInSel2=2 AND fbAnCamInDTCarryingUpDown.bInSync ) )AND
          fbCamInLeftYDUpDown.bInSync AND fbCamInLeftYDLine.bInSync  AND NOT DP_CheseCam THEN
		Ca_CanIn4:=FALSE;
		//DP_Step0:=161;
	ELSIF fbCaCamInCarryingLine2.bInSync AND fbCaCamInCarryingUpDown2.bInSync AND fbCaCamInDTCarryingLine.bInSync AND fbCaCamInDTCarryingUpDown.bInSync AND
		 fbCamInGMBuffer.bInSync AND fbCamInGMDanserMove.bInSync AND  fbCamInVirGMDriver.bInSync AND
		fbAnCamInCarryingLine.bInSync AND fbAnCamInCarryingUpDown.bInSync AND  fbAnCamInCarryingWhirling.bInSync AND  
       fbAnCamInDTCarryingLine.bInSync AND fbAnCamInDTCarryingUpDown.bInSync AND
        fbCamInLeftYDUpDown.bInSync AND fbCamInLeftYDLine.bInSync  AND DP_CheseCam THEN
		Ca_CanIn4:=FALSE;
		//DP_Step0:=161;
	END_IF		
END_IF


//
IF Ca_CanIn5 THEN   //OK
//负到正_负极搬运平移2轴凸轮耦合
	fbCaCamInCarryingLine2.ParCamIn.SlaveScaling:=1;
	fbCaCamInCarryingLine2.bCamInExecute:=TRUE;							
//负到正_负极搬运升降2轴放片凸轮耦合
	fbCaCamInCarryingUpDown2.iTableSel:=3;    //20240528SJ
	fbCaCamInCarryingUpDown2.bCamInExecute:=TRUE;					
//负到正_负极叠片平移轴凸轮耦合
	fbCaCamInDTCarryingLine.ParCamIn.SlaveScaling:=1;
	fbCaCamInDTCarryingLine.bCamInExecute:=TRUE;							
//负到正_负极叠片升降轴放片凸轮耦合
	
	fbCaCamInDTCarryingUpDown.iTableSel:=2;
	fbCaCamInDTCarryingUpDown.bCamInExecute:=TRUE;		
	
//负到正_缓存轴凸轮耦合
	fbCamInGMBuffer.iTableSel:=2;
	fbCamInGMBuffer.bCamInExecute:=TRUE;					
//负到正_隔膜平移轴凸轮耦合
	fbCamInGMDanserMove.iTableSel:=2;
	fbCamInGMDanserMove.bCamInExecute:=TRUE;

	
//负到正_放卷虚轴凸轮耦合		
	fbCamInVirGMDriver.iTableSel:=2;
	fbCamInVirGMDriver.bCamInExecute:=TRUE;		
//负到正_正极搬运平移轴凸轮耦合	
	fbAnCamInCarryingLine.ParCamIn.SlaveScaling:=-1;
	fbAnCamInCarryingLine.bCamInExecute:=TRUE;															
//负到正_正极搬运升降轴取片凸轮耦合
	fbAnCamInCarryingUpDown.iTableSel:=3;    //20240528SJ
	fbAnCamInCarryingUpDown.bCamInExecute:=TRUE;
//负到正_正极叠片平移轴凸轮耦合
	fbAnCamInDTCarryingLine.ParCamIn.SlaveScaling:=-1;
	fbAnCamInDTCarryingLine.bCamInExecute:=TRUE;	

//负到正_正极叠片升降轴取片凸轮耦合
	fbAnCamInDTCarryingUpDown.iTableSel:=3;//20240528SJ
	fbAnCamInDTCarryingUpDown.bCamInExecute:=TRUE;
//负到正_正极搬运旋转轴凸轮耦合
	fbAnCamInCarryingWhirling.ParCamIn.SlaveScaling:=-1;
	fbAnCamInCarryingWhirling.bCamInExecute:=TRUE;
//叠台左压刀升降凸轮耦合
	//fbCamInLeftYDUpDown.bCamInExecute:=TRUE;
//叠台左压刀开合凸轮耦合
	//fbCamInLeftYDLine.bCamInExecute:=TRUE;	
IF arrAxisCtrl[AxiseNo.AxisName.LeftYDLine].Cmd.arrbRealPoint[1] THEN
	fbCamInLeftYDUpDown.iTableSel:=1;
	fbCamInLeftYDLine.iTableSel:=1;
	fbCamInLeftYDUpDown.bCamInExecute:=TRUE;
	fbCamInLeftYDLine.bCamInExecute:=TRUE;	
ELSIF arrAxisCtrl[AxiseNo.AxisName.LeftYDLine].Cmd.arrbRealPoint[2] THEN	
	fbCamInLeftYDUpDown.iTableSel:=2;
	fbCamInLeftYDLine.iTableSel:=2;
	fbCamInLeftYDUpDown.bCamInExecute:=TRUE;
	fbCamInLeftYDLine.bCamInExecute:=TRUE;		
END_IF
//判断凸轮是否耦合完成
	IF fbCaCamInCarryingLine2.bInSync AND fbCaCamInDTCarryingLine.bInSync AND 
		fbCaCamInDTCarryingUpDown.bInSync  AND fbCamInGMBuffer.bInSync AND fbCamInGMDanserMove.bInSync AND
		 fbCamInVirGMDriver.bInSync AND fbAnCamInCarryingLine.bInSync AND 
		 fbCaCamInCarryingUpDown2.bInSync AND fbAnCamInCarryingUpDown.bInSync AND fbAnCamInDTCarryingUpDown.bInSync  AND 
		fbAnCamInDTCarryingLine.bInSync AND fbAnCamInCarryingWhirling.bInSync AND fbCamInLeftYDUpDown.bInSync AND
		 fbCamInLeftYDLine.bInSync  THEN
		Ca_CanIn5:=FALSE;
		//DP_Step0:=161;
	END_IF		
END_IF		

//
IF Ca_CanIn6 THEN   //OK
//负到正_负极搬运平移2轴凸轮耦合
	fbCaCamInCarryingLine2.ParCamIn.SlaveScaling:=1;
	fbCaCamInCarryingLine2.bCamInExecute:=TRUE;
//负到正_负极搬运升降2轴放片凸轮耦合
	fbCaCamInCarryingUpDown2.iTableSel:=3;  //20240528SJ
	fbCaCamInCarryingUpDown2.bCamInExecute:=TRUE;
//负到正_负极叠片平移轴凸轮耦合
	fbCaCamInDTCarryingLine.ParCamIn.SlaveScaling:=1;
	fbCaCamInDTCarryingLine.bCamInExecute:=TRUE;
//负到正_负极叠片升降轴放片凸轮耦合
	
		fbCaCamInDTCarryingUpDown.iTableSel:=2;
		fbCaCamInDTCarryingUpDown.bCamInExecute:=TRUE;
	
//叠台左压刀升降凸轮耦合
	//fbCamInLeftYDUpDown.bCamInExecute:=TRUE;
//叠台左压刀开合凸轮耦合
	//fbCamInLeftYDLine.bCamInExecute:=TRUE;	
IF arrAxisCtrl[AxiseNo.AxisName.LeftYDLine].Cmd.arrbRealPoint[1] THEN
	fbCamInLeftYDUpDown.iTableSel:=1;
	fbCamInLeftYDLine.iTableSel:=1;
	fbCamInLeftYDUpDown.bCamInExecute:=TRUE;
	fbCamInLeftYDLine.bCamInExecute:=TRUE;	
ELSIF arrAxisCtrl[AxiseNo.AxisName.LeftYDLine].Cmd.arrbRealPoint[2] THEN	
	fbCamInLeftYDUpDown.iTableSel:=2;
	fbCamInLeftYDLine.iTableSel:=2;
	fbCamInLeftYDUpDown.bCamInExecute:=TRUE;
	fbCamInLeftYDLine.bCamInExecute:=TRUE;		
END_IF
//判断凸轮耦合是否完成
	IF 	fbCaCamInCarryingLine2.bInSync AND fbCaCamInDTCarryingLine.bInSync AND 	fbCaCamInDTCarryingUpDown.bInSync  AND fbCaCamInCarryingUpDown2.bInSync AND  
		fbCamInLeftYDUpDown.bInSync AND fbCamInLeftYDLine.bInSync 	 THEN
		Ca_CanIn6:=FALSE;
		//DP_Step0:=141;
	END_IF	
END_IF		



//
IF Ca_CanIn7 THEN   //OK
//负到正_负极搬运平移2轴凸轮耦合
	fbCaCamInCarryingLine2.ParCamIn.SlaveScaling:=1;
	fbCaCamInCarryingLine2.bCamInExecute:=TRUE;						
//负到正_负极搬运升降2轴放片凸轮耦合
	fbCaCamInCarryingUpDown2.iTableSel:=3;  //20240528SJ   
	fbCaCamInCarryingUpDown2.bCamInExecute:=TRUE;
//负到正_负极叠片平移轴凸轮耦合
	fbCaCamInDTCarryingLine.ParCamIn.SlaveScaling:=1;
	fbCaCamInDTCarryingLine.bCamInExecute:=TRUE;						
//负到正_负极叠片升降轴放片凸轮耦合
		fbCaCamInDTCarryingUpDown.iTableSel:=2;
		fbCaCamInDTCarryingUpDown.bCamInExecute:=TRUE;
	
//负到正_缓存轴凸轮耦合	
	fbCamInGMBuffer.iTableSel:=2;
	fbCamInGMBuffer.bCamInExecute:=TRUE;
//负到正_隔膜平移轴凸轮耦合
	fbCamInGMDanserMove.iTableSel:=2;
	fbCamInGMDanserMove.bCamInExecute:=TRUE;

//负到正_放卷虚轴凸轮耦合
	fbCamInVirGMDriver.iTableSel:=2;
	fbCamInVirGMDriver.bCamInExecute:=TRUE;
//叠台左压刀升降凸轮耦合
	//fbCamInLeftYDUpDown.bCamInExecute:=TRUE;
//叠台左压刀开合凸轮耦合
	//fbCamInLeftYDLine.bCamInExecute:=TRUE;	
IF arrAxisCtrl[AxiseNo.AxisName.LeftYDLine].Cmd.arrbRealPoint[1] THEN
	fbCamInLeftYDUpDown.iTableSel:=1;
	fbCamInLeftYDLine.iTableSel:=1;
	fbCamInLeftYDUpDown.bCamInExecute:=TRUE;
	fbCamInLeftYDLine.bCamInExecute:=TRUE;	
ELSIF arrAxisCtrl[AxiseNo.AxisName.LeftYDLine].Cmd.arrbRealPoint[2] THEN	
	fbCamInLeftYDUpDown.iTableSel:=2;
	fbCamInLeftYDLine.iTableSel:=2;
	fbCamInLeftYDUpDown.bCamInExecute:=TRUE;
	fbCamInLeftYDLine.bCamInExecute:=TRUE;		
END_IF			
//判断凸轮耦合是否完成
	IF fbCaCamInCarryingLine2.bInSync AND fbCaCamInDTCarryingLine.bInSync AND fbCaCamInCarryingUpDown2.bInSync AND 
		fbCaCamInDTCarryingUpDown.bInSync  AND fbCamInGMBuffer.bInSync AND fbCamInGMDanserMove.bInSync AND 
		fbCamInVirGMDriver.bInSync AND fbCamInLeftYDUpDown.bInSync AND fbCamInLeftYDLine.bInSync    THEN								
			Ca_CanIn7:=FALSE;
		//DP_Step0:=141;
	END_IF
END_IF
//
IF Ca_CanIn8 THEN   //OK
//负到正_负极搬运平移2轴凸轮耦合
	fbCaCamInCarryingLine2.ParCamIn.SlaveScaling:=1;
	fbCaCamInCarryingLine2.bCamInExecute:=TRUE;
//负到正_负极搬运升降2轴放片凸轮耦合
	fbCaCamInCarryingUpDown2.iTableSel:=2;
	fbCaCamInCarryingUpDown2.bCamInExecute:=TRUE;
//负到正_负极叠片平移轴凸轮耦合
	fbCaCamInDTCarryingLine.ParCamIn.SlaveScaling:=1;
	fbCaCamInDTCarryingLine.bCamInExecute:=TRUE;
//负到正_负极叠片升降轴放片凸轮耦合
	fbCaCamInDTCarryingUpDown.iTableSel:=3;   //20240528SJ
	fbCaCamInDTCarryingUpDown.bCamInExecute:=TRUE;
//叠台左压刀升降凸轮耦合
	//fbCamInLeftYDUpDown.bCamInExecute:=TRUE;
//叠台左压刀开合凸轮耦合
	//fbCamInLeftYDLine.bCamInExecute:=TRUE;	
//判断凸轮耦合是否完成
	IF 	fbCaCamInCarryingLine2.bInSync AND fbCaCamInCarryingUpDown2	.bInSync AND 	fbCaCamInDTCarryingLine.bInSync AND fbCaCamInDTCarryingUpDown.bInSync        (*AND 	fbCaCamInDTCarryingUpDown.bInSync AND 
		fbCamInLeftYDUpDown.bInSync AND fbCamInLeftYDLine.bInSync*) 	 THEN
		Ca_CanIn8:=FALSE;
		//DP_Step0:=141;
	END_IF	
END_IF





//
IF An_CanIn1 THEN   //OK
//正到负_正极送片搬运平 移轴凸轮耦合
	fbAnCamInCarryingLine.ParCamIn.SlaveScaling:=1;
	fbAnCamInCarryingLine.bCamInExecute:=TRUE;
//正到负_正极送片搬运升降轴放片凸轮耦合
	fbAnCamInCarryingUpDown.iTableSel:=2;
	fbAnCamInCarryingUpDown.bCamInExecute:=TRUE;
//正到负_正极叠片平移轴凸轮耦合
	fbAnCamInDTCarryingLine.ParCamIn.SlaveScaling:=1;
	fbAnCamInDTCarryingLine.bCamInExecute:=TRUE;
//正到负_正极叠片升降轴放片凸轮耦合
	fbAnCamInDTCarryingUpDown.iTableSel:=2;
	fbAnCamInDTCarryingUpDown.bCamInExecute:=TRUE;
//正到负_正极搬运旋转轴凸轮耦合
fbAnCamInCarryingWhirling.ParCamIn.SlaveScaling:=1;
fbAnCamInCarryingWhirling.bCamInExecute:=TRUE;
//正到负_ 缓存轴轮耦合
	fbCamInGMBuffer.iTableSel:=1;
	 fbCamInGMBuffer.bCamInExecute:=TRUE;
//正到负_隔膜平移轴凸轮耦合
	fbCamInGMDanserMove.iTableSel:=1;
	fbCamInGMDanserMove.bCamInExecute:=TRUE;

	
//正到负_放卷虚轴凸轮耦合
	 fbCamInVirGMDriver.iTableSel :=1;
	 fbCamInVirGMDriver.bCamInExecute:=TRUE;						
//正到负_右压刀升降凸轮耦合
	//fbCamInRightYDUpDown.bCamInExecute:=TRUE;
//正极负_右压刀开合凸轮耦合
	//fbCamInRightYDLine.bCamInExecute:=TRUE;
IF arrAxisCtrl[AxiseNo.AxisName.RightYDLine].Cmd.arrbRealPoint[1] THEN	
	fbCamInRightYDUpDown.iTableSel:=1;
	fbCamInRightYDLine.iTableSel:=1;
	fbCamInRightYDUpDown.bCamInExecute:=TRUE;
    fbCamInRightYDLine.bCamInExecute:=TRUE;
ELSIF arrAxisCtrl[AxiseNo.AxisName.RightYDLine].Cmd.arrbRealPoint[2] THEN		
	fbCamInRightYDUpDown.iTableSel:=2;
	fbCamInRightYDLine.iTableSel:=2;
	fbCamInRightYDUpDown.bCamInExecute:=TRUE;
    fbCamInRightYDLine.bCamInExecute:=TRUE;	
END_IF	
//I判断凸轮耦合是否完成
	IF fbAnCamInCarryingLine.bInSync AND fbAnCamInCarryingUpDown.bInSync AND fbAnCamInDTCarryingLine.bInSync AND
		fbAnCamInDTCarryingUpDown.bInSync AND fbAnCamInCarryingWhirling.bInSync AND fbCamInGMBuffer.bInSync AND
		fbCamInGMDanserMove.bInSync AND fbCamInVirGMDriver.bInSync  AND fbCamInRightYDUpDown.bInSync AND 
		fbCamInRightYDLine.bInSync THEN
		An_CanIn1:=FALSE;
		//DP_Step0:=541;															
	END_IF					
END_IF
//
IF An_CanIn2 THEN  //OK
//正到负_正极送片搬运平移轴凸轮耦合
	fbAnCamInCarryingLine.ParCamIn.SlaveScaling:=1;
	fbAnCamInCarryingLine.bCamInExecute:=TRUE;						
//正到负_正极送片搬运升降轴放片凸轮耦合
	fbAnCamInCarryingUpDown.iTableSel:=2;
	fbAnCamInCarryingUpDown.bCamInExecute:=TRUE;
//正到负_正极叠片平移轴凸轮耦合
	fbAnCamInDTCarryingLine.ParCamIn.SlaveScaling:=1;
	fbAnCamInDTCarryingLine.bCamInExecute:=TRUE;					
//正到负_正极叠片升降轴放片凸轮耦合
	fbAnCamInDTCarryingUpDown.iTableSel:=2;
	fbAnCamInDTCarryingUpDown.bCamInExecute:=TRUE;
//正到负_正极搬运旋转轴凸轮耦合		
	fbAnCamInCarryingWhirling.ParCamIn.SlaveScaling:=1;
	fbAnCamInCarryingWhirling.bCamInExecute:=TRUE;			
//正到负_右压刀升降凸轮耦合
	//fbCamInRightYDUpDown.bCamInExecute:=TRUE;
//正极负_右压刀开合凸轮耦合
	//fbCamInRightYDLine.bCamInExecute:=TRUE;	
IF arrAxisCtrl[AxiseNo.AxisName.RightYDLine].Cmd.arrbRealPoint[1] THEN	
	fbCamInRightYDUpDown.iTableSel:=1;
	fbCamInRightYDLine.iTableSel:=1;
	fbCamInRightYDUpDown.bCamInExecute:=TRUE;
    fbCamInRightYDLine.bCamInExecute:=TRUE;
ELSIF arrAxisCtrl[AxiseNo.AxisName.RightYDLine].Cmd.arrbRealPoint[2] THEN		
	fbCamInRightYDUpDown.iTableSel:=2;
	fbCamInRightYDLine.iTableSel:=2;
	fbCamInRightYDUpDown.bCamInExecute:=TRUE;
    fbCamInRightYDLine.bCamInExecute:=TRUE;	
END_IF						 
//判断凸轮耦合是否完成
	IF fbAnCamInCarryingLine.bInSync AND fbAnCamInCarryingUpDown.bInSync AND fbAnCamInDTCarryingLine.bInSync AND fbAnCamInDTCarryingUpDown.bInSync AND 
		fbAnCamInCarryingWhirling.bInSync AND fbCamInRightYDUpDown.bInSync AND fbCamInRightYDLine.bInSync THEN
		An_CanIn2:=FALSE;
		//DP_Step0:=541;						
	END_IF			
END_IF

//
IF An_CanIn3 THEN    //OK
//正到负_正极送片搬运平移轴凸轮耦合
	fbAnCamInCarryingLine.ParCamIn.SlaveScaling:=1;
	fbAnCamInCarryingLine.bCamInExecute:=TRUE;	
//正到负_正极送片搬运升降轴放片凸轮耦合
	fbAnCamInCarryingUpDown.iTableSel:=2;
	fbAnCamInCarryingUpDown.bCamInExecute:=TRUE;
//正到负_正极叠片平移轴凸轮耦合
	fbAnCamInDTCarryingLine.ParCamIn.SlaveScaling:=1;
	fbAnCamInDTCarryingLine.bCamInExecute:=TRUE;	
//正到负_正极叠片升降轴放片凸轮耦合
	fbAnCamInDTCarryingUpDown.iTableSel:=2;
	fbAnCamInDTCarryingUpDown.bCamInExecute:=TRUE;
//正到负_正极搬运旋转轴凸轮耦合		
	fbAnCamInCarryingWhirling.ParCamIn.SlaveScaling:=1;
	fbAnCamInCarryingWhirling.bCamInExecute:=TRUE;		
//正到负_负极送片搬运平移轴凸轮耦合
	fbCaCamInCarryingLine2.ParCamIn.SlaveScaling:=-1;
	fbCaCamInCarryingLine2.bCamInExecute:=TRUE;
	
//正到负_负极送片搬运升降轴取片凸轮耦合 
  IF Mach_Control.U.EmptyRunMode THEN
	 fbCaCamInCarryingUpDown2.iTableSel:=3;
	 fbCaCamInCarryingUpDown2.bCamInExecute:=TRUE;//20240509 CF    //20240528SJ   NOT Mach_Control.U.EmptyRunMode
  ELSE
	 fbCaCamInCarryingUpDown2.iTableSel:=1;
	 fbCaCamInCarryingUpDown2.bCamInExecute:=TRUE;//20240509 CF    //20240528SJ   NOT Mach_Control.U.EmptyRunMode	  
  END_IF
	 
	 
//正到负_负极叠片搬运平移轴凸轮耦合
	fbCaCamInDTCarryingLine.ParCamIn.SlaveScaling:=-1;
	fbCaCamInDTCarryingLine.bCamInExecute:=TRUE;
//正到负_负极叠片搬运升降轴取片凸轮耦合
	fbCaCamInDTCarryingUpDown.iTableSel:=1;
	fbCaCamInDTCarryingUpDown.bCamInExecute:=TRUE;
//正到负_负极叠片搬运升降轴取片凸轮耦合
	IF iCaCamInSel2=1 THEN
		fbCaCamInDTCarryingUpDown.iTableSel:=1;
		fbCaCamInDTCarryingUpDown.bCamInExecute:=TRUE;
	END_IF	
//正到负_ 缓存轴轮耦合
	fbCamInGMBuffer.iTableSel:=1;
	 fbCamInGMBuffer.bCamInExecute:=TRUE;
//正到负_隔膜平移轴凸轮耦合
	fbCamInGMDanserMove.iTableSel:=1;
	fbCamInGMDanserMove.bCamInExecute:=TRUE;
	


